LIN {X 0,Y 368.346,Z 298.483,A -85,B 0,C 180,E1 -13235.936,E2 -13235.936} C_VEL
LIN {X 0,Y 372.9,Z 313.274,A -85,B 0,C 180,E1 -13237.03,E2 -13237.03} C_VEL
LIN {X 0,Y 374.658,Z 319.531,A -85,B 0,C 180,E1 -13237.544,E2 -13237.544} C_VEL
LIN {X 0,Y 373.455,Z 332.306,A -85,B 0,C 180,E1 -13238.385,E2 -13238.385} C_VEL
LIN {X 0,Y 371.968,Z 346.016,A -85,B 0,C 180,E1 -13239.515,E2 -13239.515} C_VEL
LIN {X 0,Y 370.336,Z 358.794,A -85,B 0,C 180,E1 -13240.804,E2 -13240.804} C_VEL
LIN {X 0,Y 368.69,Z 371.331,A -85,B 0,C 180,E1 -13242.352,E2 -13242.352} C_VEL
LIN {X 0,Y 366.908,Z 383.259,A -85,B 0,C 180,E1 -13244.135,E2 -13244.135} C_VEL
LIN {X 0,Y 365.422,Z 393.227,A -85,B 0,C 180,E1 -13245.931,E2 -13245.931} C_VEL
LIN {X 0,Y 363.933,Z 402.704,A -85,B 0,C 180,E1 -13247.997,E2 -13247.997} C_VEL
LIN {X 0,Y 362.831,Z 410.613,A -85,B 0,C 180,E1 -13250.109,E2 -13250.109} C_VEL
LIN {X 0,Y 361.936,Z 417.12,A -85,B 0,C 180,E1 -13252.249,E2 -13252.249} C_VEL
LIN {X 0,Y 361.391,Z 421.607,A -85,B 0,C 180,E1 -13254.103,E2 -13254.103} C_VEL
LIN {X 0,Y 360.855,Z 426.279,A -85,B 0,C 180,E1 -13256.611,E2 -13256.611} C_VEL
LIN {X 0,Y 360.458,Z 429.462,A -85,B 0,C 180,E1 -13259.171,E2 -13259.171} C_VEL
LIN {X 0,Y 360.358,Z 430.738,A -85,B 0,C 180,E1 -13260.897,E2 -13260.897} C_VEL
LIN {X 0,Y 360.322,Z 431.406,A -85,B 0,C 180,E1 -13263.101,E2 -13263.101} C_VEL
LIN {X 0,Y 360.359,Z 431.048,A -85,B 0,C 180,E1 -13265.007,E2 -13265.007} C_VEL
LIN {X 0,Y 360.534,Z 429.695,A -85,B 0,C 180,E1 -13267.177,E2 -13267.177} C_VEL
LIN {X 0,Y 360.574,Z 429.284,A -85,B 0,C 180,E1 -13267.57,E2 -13267.57} C_VEL
LIN {X 0,Y 360.044,Z 428.403,A -85,B 0,C 180,E1 -13268.493,E2 -13268.493} C_VEL
LIN {X 0,Y 357.472,Z 426.615,A -85,B 0,C 180,E1 -13269.998,E2 -13269.998} C_VEL
LIN {X 0,Y 355.343,Z 424.907,A -85,B 0,C 180,E1 -13271.203,E2 -13271.203} C_VEL
LIN {X 0,Y 354.556,Z 423.304,A -85,B 0,C 180,E1 -13272.116,E2 -13272.116} C_VEL
LIN {X 0,Y 354.562,Z 422.675,A -85,B 0,C 180,E1 -13272.42,E2 -13272.42} C_VEL
LIN {X 0,Y 355.32,Z 417.558,A -85,B 0,C 180,E1 -13274.6,E2 -13274.6} C_VEL
LIN {X 0,Y 356.455,Z 410.865,A -85,B 0,C 180,E1 -13276.844,E2 -13276.844} C_VEL
LIN {X 0,Y 357.829,Z 402.794,A -85,B 0,C 180,E1 -13279.018,E2 -13279.018} C_VEL
LIN {X 0,Y 359.353,Z 394.035,A -85,B 0,C 180,E1 -13280.959,E2 -13280.959} C_VEL
LIN {X 0,Y 361.095,Z 384.034,A -85,B 0,C 180,E1 -13282.795,E2 -13282.795} C_VEL
LIN {X 0,Y 362.941,Z 372.942,A -85,B 0,C 180,E1 -13284.487,E2 -13284.487} C_VEL
LIN {X 0,Y 364.899,Z 360.545,A -85,B 0,C 180,E1 -13286.047,E2 -13286.047} C_VEL
LIN {X 0,Y 366.644,Z 347.802,A -85,B 0,C 180,E1 -13287.373,E2 -13287.373} C_VEL
LIN {X 0,Y 368.422,Z 333.632,A -85,B 0,C 180,E1 -13288.556,E2 -13288.556} C_VEL
LIN {X 0,Y 369.441,Z 323.375,A -85,B 0,C 180,E1 -13289.254,E2 -13289.254} C_VEL
LIN {X 0,Y 365.365,Z 309.416,A -85,B 0,C 180,E1 -13290.491,E2 -13290.491} C_VEL
LIN {X 0,Y 359.944,Z 295.452,A -85,B 0,C 180,E1 -13291.663,E2 -13291.663} C_VEL
LIN {X 0,Y 355.644,Z 286.065,A -85,B 0,C 180,E1 -13292.411,E2 -13292.411} C_VEL
LIN {X 0,Y 354.613,Z 283.116,A -85,B 0,C 180,E1 -13292.604,E2 -13292.604} C_VEL
LIN {X 0,Y 354.73,Z 280.957,A -85,B 0,C 180,E1 -13295.692,E2 -13295.692} C_VEL
LIN {X 0,Y 354.874,Z 278.678,A -85,B 0,C 180,E1 -13299.118,E2 -13299.118} C_VEL
LIN {X 0,Y 354.894,Z 276.415,A -85,B 0,C 180,E1 -13302.721,E2 -13302.721} C_VEL
LIN {X 0,Y 354.867,Z 275.912,A -85,B 0,C 180,E1 -13303.904,E2 -13303.904} C_VEL
LIN {X 0,Y 354.915,Z 275.902,A -85,B 0,C 180,E1 -13307.42,E2 -13307.42} C_VEL
LIN {X 0,Y 355.122,Z 275.877,A -85,B 0,C 180,E1 -13311.69,E2 -13311.69} C_VEL
LIN {X 0,Y 355.088,Z 275.879,A -85,B 0,C 180,E1 -13314.322,E2 -13314.322} C_VEL
LIN {X 0,Y 355.241,Z 275.859,A -85,B 0,C 180,E1 -13317.734,E2 -13317.734} C_VEL
LIN {X 0,Y 355.393,Z 275.839,A -85,B 0,C 180,E1 -13320.001,E2 -13320.001} C_VEL
LIN {X 0,Y 355.242,Z 275.858,A -85,B 0,C 180,E1 -13322.269,E2 -13322.269} C_VEL
LIN {X 0,Y 355.134,Z 275.873,A -85,B 0,C 180,E1 -13326.82,E2 -13326.82} C_VEL
LIN {X 0,Y 355.011,Z 275.888,A -85,B 0,C 180,E1 -13329.114,E2 -13329.114} C_VEL
LIN {X 0,Y 354.918,Z 275.898,A -85,B 0,C 180,E1 -13332.582,E2 -13332.582} C_VEL
LIN {X 0,Y 354.886,Z 275.904,A -85,B 0,C 180,E1 -13336.097,E2 -13336.097} C_VEL
LIN {X 0,Y 354.903,Z 275.902,A -85,B 0,C 180,E1 -13338.473,E2 -13338.473} C_VEL
LIN {X 0,Y 354.832,Z 275.911,A -85,B 0,C 180,E1 -13342.107,E2 -13342.107} C_VEL
LIN {X 0,Y 354.897,Z 275.902,A -85,B 0,C 180,E1 -13345.829,E2 -13345.829} C_VEL
LIN {X 0,Y 354.852,Z 275.914,A -85,B 0,C 180,E1 -13349.68,E2 -13349.68} C_VEL
LIN {X 0,Y 354.82,Z 276.044,A -85,B 0,C 180,E1 -13352.667,E2 -13352.667} C_VEL
LIN {X 0,Y 355.388,Z 279.05,A -85,B 0,C 180,E1 -13355.828,E2 -13355.828} C_VEL
LIN {X 0,Y 356.119,Z 283.281,A -85,B 0,C 180,E1 -13359.678,E2 -13359.678} C_VEL
LIN {X 0,Y 356.952,Z 288.147,A -85,B 0,C 180,E1 -13363.561,E2 -13363.561} C_VEL
LIN {X 0,Y 357.671,Z 292.442,A -85,B 0,C 180,E1 -13366.639,E2 -13366.639} C_VEL
LIN {X 0,Y 357.676,Z 295.963,A -85,B 0,C 180,E1 -13368.935,E2 -13368.935} C_VEL
LIN {X 0,Y 356.892,Z 301.707,A -85,B 0,C 180,E1 -13372.378,E2 -13372.378} C_VEL
LIN {X 0,Y 356.195,Z 308.035,A -85,B 0,C 180,E1 -13375.966,E2 -13375.966} C_VEL
LIN {X 0,Y 355.518,Z 315.02,A -85,B 0,C 180,E1 -13379.73,E2 -13379.73} C_VEL
LIN {X 0,Y 355.426,Z 316.517,A -85,B 0,C 180,E1 -13380.464,E2 -13380.464} C_VEL
LIN {X 0,Y 356.367,Z 319.81,A -85,B 0,C 180,E1 -13380.638,E2 -13380.638} C_VEL
LIN {X 0,Y 360.801,Z 334.796,A -85,B 0,C 180,E1 -13381.548,E2 -13381.548} C_VEL
LIN {X 0,Y 364.028,Z 349.7,A -85,B 0,C 180,E1 -13382.552,E2 -13382.552} C_VEL
LIN {X 0,Y 366.315,Z 364.769,A -85,B 0,C 180,E1 -13383.695,E2 -13383.695} C_VEL
LIN {X 0,Y 367.111,Z 371.055,A -85,B 0,C 180,E1 -13384.231,E2 -13384.231} C_VEL
LIN {X 0,Y 365.414,Z 384.335,A -85,B 0,C 180,E1 -13385.273,E2 -13385.273} C_VEL
LIN {X 0,Y 363.482,Z 397.146,A -85,B 0,C 180,E1 -13386.498,E2 -13386.498} C_VEL
LIN {X 0,Y 361.493,Z 410.148,A -85,B 0,C 180,E1 -13388.023,E2 -13388.023} C_VEL
LIN {X 0,Y 359.534,Z 422.392,A -85,B 0,C 180,E1 -13389.766,E2 -13389.766} C_VEL
LIN {X 0,Y 357.871,Z 433.506,A -85,B 0,C 180,E1 -13391.688,E2 -13391.688} C_VEL
LIN {X 0,Y 356.341,Z 443.099,A -85,B 0,C 180,E1 -13393.678,E2 -13393.678} C_VEL
LIN {X 0,Y 355.149,Z 451.18,A -85,B 0,C 180,E1 -13395.698,E2 -13395.698} C_VEL
LIN {X 0,Y 354.343,Z 458.64,A -85,B 0,C 180,E1 -13397.981,E2 -13397.981} C_VEL
LIN {X 0,Y 353.715,Z 464.622,A -85,B 0,C 180,E1 -13400.278,E2 -13400.278} C_VEL
LIN {X 0,Y 353.51,Z 468.2,A -85,B 0,C 180,E1 -13402.001,E2 -13402.001} C_VEL
LIN {X 0,Y 353.366,Z 471.82,A -85,B 0,C 180,E1 -13404.294,E2 -13404.294} C_VEL
LIN {X 0,Y 353.27,Z 474.207,A -85,B 0,C 180,E1 -13406.579,E2 -13406.579} C_VEL
LIN {X 0,Y 353.379,Z 475.424,A -85,B 0,C 180,E1 -13408.861,E2 -13408.861} C_VEL
LIN {X 0,Y 353.378,Z 475.45,A -85,B 0,C 180,E1 -13411.14,E2 -13411.14} C_VEL
LIN {X 0,Y 353.261,Z 474.249,A -85,B 0,C 180,E1 -13413.422,E2 -13413.422} C_VEL
LIN {X 0,Y 353.358,Z 471.874,A -85,B 0,C 180,E1 -13415.708,E2 -13415.708} C_VEL
LIN {X 0,Y 353.511,Z 468.264,A -85,B 0,C 180,E1 -13418,E2 -13418} C_VEL
LIN {X 0,Y 353.821,Z 463.331,A -85,B 0,C 180,E1 -13420.299,E2 -13420.299} C_VEL
LIN {X 0,Y 354.511,Z 456.958,A -85,B 0,C 180,E1 -13422.596,E2 -13422.596} C_VEL
LIN {X 0,Y 355.5,Z 448.962,A -85,B 0,C 180,E1 -13424.893,E2 -13424.893} C_VEL
LIN {X 0,Y 356.729,Z 440.46,A -85,B 0,C 180,E1 -13426.894,E2 -13426.894} C_VEL
LIN {X 0,Y 358.097,Z 431.831,A -85,B 0,C 180,E1 -13428.599,E2 -13428.599} C_VEL
LIN {X 0,Y 359.718,Z 420.925,A -85,B 0,C 180,E1 -13430.41,E2 -13430.41} C_VEL
LIN {X 0,Y 361.661,Z 408.477,A -85,B 0,C 180,E1 -13432.118,E2 -13432.118} C_VEL
LIN {X 0,Y 363.565,Z 394.852,A -85,B 0,C 180,E1 -13433.649,E2 -13433.649} C_VEL
LIN {X 0,Y 365.524,Z 381.257,A -85,B 0,C 180,E1 -13434.873,E2 -13434.873} C_VEL
LIN {X 0,Y 366.729,Z 369.526,A -85,B 0,C 180,E1 -13435.748,E2 -13435.748} C_VEL
LIN {X 0,Y 364.294,Z 355.037,A -85,B 0,C 180,E1 -13436.879,E2 -13436.879} C_VEL
LIN {X 0,Y 361.413,Z 340.742,A -85,B 0,C 180,E1 -13437.821,E2 -13437.821} C_VEL
LIN {X 0,Y 357.374,Z 325.464,A -85,B 0,C 180,E1 -13438.689,E2 -13438.689} C_VEL
LIN {X 0,Y 355.389,Z 318.138,A -85,B 0,C 180,E1 -13439.057,E2 -13439.057} C_VEL
LIN {X 0,Y 355.926,Z 312.143,A -85,B 0,C 180,E1 -13442.218,E2 -13442.218} C_VEL
LIN {X 0,Y 356.589,Z 306.081,A -85,B 0,C 180,E1 -13445.488,E2 -13445.488} C_VEL
LIN {X 0,Y 357.325,Z 299.823,A -85,B 0,C 180,E1 -13449.006,E2 -13449.006} C_VEL
LIN {X 0,Y 357.761,Z 294.883,A -85,B 0,C 180,E1 -13451.907,E2 -13451.907} C_VEL
LIN {X 0,Y 357.548,Z 291.222,A -85,B 0,C 180,E1 -13454.2,E2 -13454.2} C_VEL
LIN {X 0,Y 356.56,Z 285.705,A -85,B 0,C 180,E1 -13457.92,E2 -13457.92} C_VEL
LIN {X 0,Y 355.823,Z 281.709,A -85,B 0,C 180,E1 -13460.798,E2 -13460.798} C_VEL
LIN {X 0,Y 355.104,Z 277.225,A -85,B 0,C 180,E1 -13464.238,E2 -13464.238} C_VEL
LIN {X 0,Y 354.843,Z 275.911,A -85,B 0,C 180,E1 -13465.462,E2 -13465.462} C_VEL
LIN {X 0,Y 354.806,Z 275.915,A -85,B 0,C 180,E1 -13469.001,E2 -13469.001} C_VEL
LIN {X 0,Y 354.888,Z 275.905,A -85,B 0,C 180,E1 -13472.903,E2 -13472.903} C_VEL
LIN {X 0,Y 354.867,Z 275.903,A -85,B 0,C 180,E1 -13475.647,E2 -13475.647} C_VEL
LIN {X 0,Y 354.846,Z 275.908,A -85,B 0,C 180,E1 -13479.113,E2 -13479.113} C_VEL
LIN {X 0,Y 354.904,Z 275.904,A -85,B 0,C 180,E1 -13482.719,E2 -13482.719} C_VEL
LIN {X 0,Y 354.957,Z 275.894,A -85,B 0,C 180,E1 -13486.254,E2 -13486.254} C_VEL
LIN {X 0,Y 354.983,Z 275.889,A -85,B 0,C 180,E1 -13489.735,E2 -13489.735} C_VEL
LIN {X 0,Y 355.105,Z 275.874,A -85,B 0,C 180,E1 -13493.179,E2 -13493.179} C_VEL
LIN {X 0,Y 355.248,Z 275.856,A -85,B 0,C 180,E1 -13497.731,E2 -13497.731} C_VEL
LIN {X 0,Y 355.402,Z 275.838,A -85,B 0,C 180,E1 -13499.999,E2 -13499.999} C_VEL
LIN {X 0,Y 355.247,Z 275.86,A -85,B 0,C 180,E1 -13502.266,E2 -13502.266} C_VEL
LIN {X 0,Y 355.142,Z 275.87,A -85,B 0,C 180,E1 -13506.818,E2 -13506.818} C_VEL
LIN {X 0,Y 355.018,Z 275.884,A -85,B 0,C 180,E1 -13509.111,E2 -13509.111} C_VEL
LIN {X 0,Y 354.924,Z 275.898,A -85,B 0,C 180,E1 -13512.579,E2 -13512.579} C_VEL
LIN {X 0,Y 354.892,Z 275.905,A -85,B 0,C 180,E1 -13516.094,E2 -13516.094} C_VEL
LIN {X 0,Y 354.908,Z 275.9,A -85,B 0,C 180,E1 -13518.47,E2 -13518.47} C_VEL
LIN {X 0,Y 354.835,Z 275.912,A -85,B 0,C 180,E1 -13522.104,E2 -13522.104} C_VEL
LIN {X 0,Y 354.899,Z 275.902,A -85,B 0,C 180,E1 -13525.826,E2 -13525.826} C_VEL
LIN {X 0,Y 354.816,Z 275.911,A -85,B 0,C 180,E1 -13529.68,E2 -13529.68} C_VEL
LIN {X 0,Y 354.804,Z 275.914,A -85,B 0,C 180,E1 -13533.7,E2 -13533.7} C_VEL
LIN {X 0,Y 354.796,Z 275.913,A -85,B 0,C 180,E1 -13536.458,E2 -13536.458} C_VEL
LIN {X 0,Y 354.821,Z 275.91,A -85,B 0,C 180,E1 -13539.422,E2 -13539.422} C_VEL
LIN {X 0,Y 354.788,Z 275.912,A -85,B 0,C 180,E1 -13542.866,E2 -13542.866} C_VEL
LIN {X 0,Y 354.848,Z 275.908,A -85,B 0,C 180,E1 -13546.115,E2 -13546.115} C_VEL
LIN {X 0,Y 354.852,Z 275.905,A -85,B 0,C 180,E1 -13549.187,E2 -13549.187} C_VEL
LIN {X 0,Y 354.803,Z 275.911,A -85,B 0,C 180,E1 -13552.401,E2 -13552.401} C_VEL
LIN {X 0,Y 354.806,Z 275.91,A -85,B 0,C 180,E1 -13554.939,E2 -13554.939} C_VEL
LIN {X 0,Y 354.786,Z 275.913,A -85,B 0,C 180,E1 -13558.404,E2 -13558.404} C_VEL
LIN {X 0,Y 354.846,Z 275.912,A -85,B 0,C 180,E1 -13561.618,E2 -13561.618} C_VEL
LIN {X 0,Y 354.891,Z 275.901,A -85,B 0,C 180,E1 -13564.171,E2 -13564.171} C_VEL
LIN {X 0,Y 354.826,Z 275.91,A -85,B 0,C 180,E1 -13567.893,E2 -13567.893} C_VEL
LIN {X 0,Y 354.914,Z 275.899,A -85,B 0,C 180,E1 -13571.89,E2 -13571.89} C_VEL
LIN {X 0,Y 354.934,Z 275.896,A -85,B 0,C 180,E1 -13575.98,E2 -13575.98} C_VEL
LIN {X 0,Y 354.973,Z 275.892,A -85,B 0,C 180,E1 -13579.735,E2 -13579.735} C_VEL
LIN {X 0,Y 355.103,Z 275.873,A -85,B 0,C 180,E1 -13582.036,E2 -13582.036} C_VEL
LIN {X 0,Y 355.066,Z 275.878,A -85,B 0,C 180,E1 -13584.32,E2 -13584.32} C_VEL
LIN {X 0,Y 355.015,Z 276.113,A -85,B 0,C 180,E1 -13588.865,E2 -13588.865} C_VEL
LIN {X 0,Y 354.385,Z 280.472,A -85,B 0,C 180,E1 -13594.193,E2 -13594.193} C_VEL
LIN {X 0,Y 356.694,Z 286.53,A -85,B 0,C 180,E1 -13594.558,E2 -13594.558} C_VEL
LIN {X 0,Y 362.27,Z 301.422,A -85,B 0,C 180,E1 -13595.587,E2 -13595.587} C_VEL
LIN {X 0,Y 366.282,Z 314.648,A -85,B 0,C 180,E1 -13596.61,E2 -13596.61} C_VEL
LIN {X 0,Y 368.088,Z 321.326,A -85,B 0,C 180,E1 -13597.179,E2 -13597.179} C_VEL
LIN {X 0,Y 366.7,Z 334.988,A -85,B 0,C 180,E1 -13598.125,E2 -13598.125} C_VEL
LIN {X 0,Y 365.203,Z 348.245,A -85,B 0,C 180,E1 -13599.274,E2 -13599.274} C_VEL
LIN {X 0,Y 363.578,Z 360.207,A -85,B 0,C 180,E1 -13600.524,E2 -13600.524} C_VEL
LIN {X 0,Y 361.934,Z 372.216,A -85,B 0,C 180,E1 -13602.048,E2 -13602.048} C_VEL
LIN {X 0,Y 360.447,Z 382.067,A -85,B 0,C 180,E1 -13603.53,E2 -13603.53} C_VEL
LIN {X 0,Y 358.81,Z 392.168,A -85,B 0,C 180,E1 -13605.332,E2 -13605.332} C_VEL
LIN {X 0,Y 357.39,Z 400.719,A -85,B 0,C 180,E1 -13607.155,E2 -13607.155} C_VEL
LIN {X 0,Y 356.256,Z 408.565,A -85,B 0,C 180,E1 -13609.166,E2 -13609.166} C_VEL
LIN {X 0,Y 355.443,Z 414.117,A -85,B 0,C 180,E1 -13610.848,E2 -13610.848} C_VEL
LIN {X 0,Y 354.704,Z 419.222,A -85,B 0,C 180,E1 -13612.728,E2 -13612.728} C_VEL
LIN {X 0,Y 354.179,Z 423.45,A -85,B 0,C 180,E1 -13614.626,E2 -13614.626} C_VEL
LIN {X 0,Y 353.78,Z 426.91,A -85,B 0,C 180,E1 -13616.631,E2 -13616.631} C_VEL
LIN {X 0,Y 353.408,Z 429.74,A -85,B 0,C 180,E1 -13618.959,E2 -13618.959} C_VEL
LIN {X 0,Y 353.273,Z 431.32,A -85,B 0,C 180,E1 -13621.195,E2 -13621.195} C_VEL
LIN {X 0,Y 353.226,Z 431.845,A -85,B 0,C 180,E1 -13623.319,E2 -13623.319} C_VEL
LIN {X 0,Y 353.284,Z 431.388,A -85,B 0,C 180,E1 -13625.354,E2 -13625.354} C_VEL
LIN {X 0,Y 353.575,Z 429.439,A -85,B 0,C 180,E1 -13628.037,E2 -13628.037} C_VEL
LIN {X 0,Y 353.97,Z 426.681,A -85,B 0,C 180,E1 -13630.185,E2 -13630.185} C_VEL
LIN {X 0,Y 354.562,Z 422.675,A -85,B 0,C 180,E1 -13632.42,E2 -13632.42} C_VEL
LIN {X 0,Y 354.187,Z 420.817,A -85,B 0,C 180,E1 -13633.324,E2 -13633.324} C_VEL
LIN {X 0,Y 351.901,Z 417.626,A -85,B 0,C 180,E1 -13634.804,E2 -13634.804} C_VEL
LIN {X 0,Y 349.743,Z 413.979,A -85,B 0,C 180,E1 -13636.27,E2 -13636.27} C_VEL
LIN {X 0,Y 349.567,Z 411.346,A -85,B 0,C 180,E1 -13637.137,E2 -13637.137} C_VEL
LIN {X 0,Y 350.959,Z 403.72,A -85,B 0,C 180,E1 -13639.25,E2 -13639.25} C_VEL
LIN {X 0,Y 352.567,Z 394.833,A -85,B 0,C 180,E1 -13641.271,E2 -13641.271} C_VEL
LIN {X 0,Y 354.314,Z 385.25,A -85,B 0,C 180,E1 -13643.079,E2 -13643.079} C_VEL
LIN {X 0,Y 356.349,Z 373.692,A -85,B 0,C 180,E1 -13644.89,E2 -13644.89} C_VEL
LIN {X 0,Y 358.349,Z 361.629,A -85,B 0,C 180,E1 -13646.446,E2 -13646.446} C_VEL
LIN {X 0,Y 360.282,Z 348.202,A -85,B 0,C 180,E1 -13647.871,E2 -13647.871} C_VEL
LIN {X 0,Y 362.13,Z 334.183,A -85,B 0,C 180,E1 -13649.058,E2 -13649.058} C_VEL
LIN {X 0,Y 362.94,Z 326.406,A -85,B 0,C 180,E1 -13649.612,E2 -13649.612} C_VEL
LIN {X 0,Y 362.56,Z 323.397,A -85,B 0,C 180,E1 -13649.863,E2 -13649.863} C_VEL
LIN {X 0,Y 358.992,Z 311.346,A -85,B 0,C 180,E1 -13650.983,E2 -13650.983} C_VEL
LIN {X 0,Y 354.258,Z 298.775,A -85,B 0,C 180,E1 -13652.093,E2 -13652.093} C_VEL
LIN {X 0,Y 349.013,Z 287.122,A -85,B 0,C 180,E1 -13653.067,E2 -13653.067} C_VEL
LIN {X 0,Y 347.779,Z 284.415,A -85,B 0,C 180,E1 -13653.285,E2 -13653.285} C_VEL
LIN {X 0,Y 347.631,Z 283.617,A -85,B 0,C 180,E1 -13653.353,E2 -13653.353} C_VEL
LIN {X 0,Y 347.713,Z 281.728,A -85,B 0,C 180,E1 -13656.158,E2 -13656.158} C_VEL
LIN {X 0,Y 347.854,Z 280.077,A -85,B 0,C 180,E1 -13658.676,E2 -13658.676} C_VEL
LIN {X 0,Y 347.901,Z 277.805,A -85,B 0,C 180,E1 -13662.363,E2 -13662.363} C_VEL
LIN {X 0,Y 347.853,Z 276.785,A -85,B 0,C 180,E1 -13664.774,E2 -13664.774} C_VEL
LIN {X 0,Y 347.878,Z 276.778,A -85,B 0,C 180,E1 -13668.346,E2 -13668.346} C_VEL
LIN {X 0,Y 348.068,Z 276.756,A -85,B 0,C 180,E1 -13671.876,E2 -13671.876} C_VEL
LIN {X 0,Y 348.063,Z 276.754,A -85,B 0,C 180,E1 -13674.207,E2 -13674.207} C_VEL
LIN {X 0,Y 348.204,Z 276.735,A -85,B 0,C 180,E1 -13677.688,E2 -13677.688} C_VEL
LIN {X 0,Y 348.342,Z 276.717,A -85,B 0,C 180,E1 -13680.001,E2 -13680.001} C_VEL
LIN {X 0,Y 348.204,Z 276.735,A -85,B 0,C 180,E1 -13682.315,E2 -13682.315} C_VEL
LIN {X 0,Y 348.103,Z 276.749,A -85,B 0,C 180,E1 -13686.959,E2 -13686.959} C_VEL
LIN {X 0,Y 347.964,Z 276.767,A -85,B 0,C 180,E1 -13689.3,E2 -13689.3} C_VEL
LIN {X 0,Y 347.887,Z 276.772,A -85,B 0,C 180,E1 -13692.841,E2 -13692.841} C_VEL
LIN {X 0,Y 347.836,Z 276.782,A -85,B 0,C 180,E1 -13696.433,E2 -13696.433} C_VEL
LIN {X 0,Y 347.853,Z 276.779,A -85,B 0,C 180,E1 -13698.861,E2 -13698.861} C_VEL
LIN {X 0,Y 347.772,Z 276.792,A -85,B 0,C 180,E1 -13702.581,E2 -13702.581} C_VEL
LIN {X 0,Y 347.81,Z 276.784,A -85,B 0,C 180,E1 -13705.11,E2 -13705.11} C_VEL
LIN {X 0,Y 347.809,Z 276.787,A -85,B 0,C 180,E1 -13707.695,E2 -13707.695} C_VEL
LIN {X 0,Y 347.762,Z 276.796,A -85,B 0,C 180,E1 -13710.348,E2 -13710.348} C_VEL
LIN {X 0,Y 347.797,Z 277.037,A -85,B 0,C 180,E1 -13711.931,E2 -13711.931} C_VEL
LIN {X 0,Y 348.458,Z 280.588,A -85,B 0,C 180,E1 -13715.797,E2 -13715.797} C_VEL
LIN {X 0,Y 348.956,Z 283.6,A -85,B 0,C 180,E1 -13718.635,E2 -13718.635} C_VEL
LIN {X 0,Y 349.619,Z 287.493,A -85,B 0,C 180,E1 -13721.948,E2 -13721.948} C_VEL
LIN {X 0,Y 350.464,Z 292.031,A -85,B 0,C 180,E1 -13725.424,E2 -13725.424} C_VEL
LIN {X 0,Y 350.758,Z 295.538,A -85,B 0,C 180,E1 -13727.848,E2 -13727.848} C_VEL
LIN {X 0,Y 350.227,Z 300.199,A -85,B 0,C 180,E1 -13730.795,E2 -13730.795} C_VEL
LIN {X 0,Y 349.499,Z 306.156,A -85,B 0,C 180,E1 -13734.328,E2 -13734.328} C_VEL
LIN {X 0,Y 348.775,Z 312.345,A -85,B 0,C 180,E1 -13737.815,E2 -13737.815} C_VEL
LIN {X 0,Y 348.47,Z 315.987,A -85,B 0,C 180,E1 -13739.748,E2 -13739.748} C_VEL
LIN {X 0,Y 349.445,Z 319.338,A -85,B 0,C 180,E1 -13739.938,E2 -13739.938} C_VEL
LIN {X 0,Y 354.287,Z 335.29,A -85,B 0,C 180,E1 -13740.973,E2 -13740.973} C_VEL
LIN {X 0,Y 357.541,Z 350.356,A -85,B 0,C 180,E1 -13742.031,E2 -13742.031} C_VEL
LIN {X 0,Y 359.836,Z 366.392,A -85,B 0,C 180,E1 -13743.308,E2 -13743.308} C_VEL
LIN {X 0,Y 360.556,Z 372.164,A -85,B 0,C 180,E1 -13743.823,E2 -13743.823} C_VEL
LIN {X 0,Y 358.716,Z 385.725,A -85,B 0,C 180,E1 -13744.934,E2 -13744.934} C_VEL
LIN {X 0,Y 356.54,Z 399.492,A -85,B 0,C 180,E1 -13746.321,E2 -13746.321} C_VEL
LIN {X 0,Y 354.483,Z 412.02,A -85,B 0,C 180,E1 -13747.872,E2 -13747.872} C_VEL
LIN {X 0,Y 352.44,Z 424.352,A -85,B 0,C 180,E1 -13749.725,E2 -13749.725} C_VEL
LIN {X 0,Y 350.789,Z 434.671,A -85,B 0,C 180,E1 -13751.607,E2 -13751.607} C_VEL
LIN {X 0,Y 349.275,Z 443.978,A -85,B 0,C 180,E1 -13753.639,E2 -13753.639} C_VEL
LIN {X 0,Y 347.964,Z 452.21,A -85,B 0,C 180,E1 -13755.81,E2 -13755.81} C_VEL
LIN {X 0,Y 347.32,Z 458.229,A -85,B 0,C 180,E1 -13757.734,E2 -13757.734} C_VEL
LIN {X 0,Y 346.657,Z 464.204,A -85,B 0,C 180,E1 -13760.078,E2 -13760.078} C_VEL
LIN {X 0,Y 346.43,Z 467.782,A -85,B 0,C 180,E1 -13761.837,E2 -13761.837} C_VEL
LIN {X 0,Y 346.291,Z 471.396,A -85,B 0,C 180,E1 -13764.177,E2 -13764.177} C_VEL
LIN {X 0,Y 346.192,Z 473.777,A -85,B 0,C 180,E1 -13766.509,E2 -13766.509} C_VEL
LIN {X 0,Y 346.301,Z 474.987,A -85,B 0,C 180,E1 -13768.838,E2 -13768.838} C_VEL
LIN {X 0,Y 346.301,Z 475.011,A -85,B 0,C 180,E1 -13771.164,E2 -13771.164} C_VEL
LIN {X 0,Y 346.184,Z 473.799,A -85,B 0,C 180,E1 -13773.492,E2 -13773.492} C_VEL
LIN {X 0,Y 346.328,Z 471.085,A -85,B 0,C 180,E1 -13776.087,E2 -13776.087} C_VEL
LIN {X 0,Y 346.499,Z 466.706,A -85,B 0,C 180,E1 -13778.751,E2 -13778.751} C_VEL
LIN {X 0,Y 346.951,Z 461.396,A -85,B 0,C 180,E1 -13781.096,E2 -13781.096} C_VEL
LIN {X 0,Y 347.726,Z 454.615,A -85,B 0,C 180,E1 -13783.441,E2 -13783.441} C_VEL
LIN {X 0,Y 348.718,Z 447.312,A -85,B 0,C 180,E1 -13785.489,E2 -13785.489} C_VEL
LIN {X 0,Y 350.024,Z 438.551,A -85,B 0,C 180,E1 -13787.529,E2 -13787.529} C_VEL
LIN {X 0,Y 351.806,Z 428.034,A -85,B 0,C 180,E1 -13789.55,E2 -13789.55} C_VEL
LIN {X 0,Y 353.456,Z 417.252,A -85,B 0,C 180,E1 -13791.278,E2 -13791.278} C_VEL
LIN {X 0,Y 355.535,Z 404.358,A -85,B 0,C 180,E1 -13792.98,E2 -13792.98} C_VEL
LIN {X 0,Y 357.427,Z 391.353,A -85,B 0,C 180,E1 -13794.389,E2 -13794.389} C_VEL
LIN {X 0,Y 359.477,Z 377.334,A -85,B 0,C 180,E1 -13795.606,E2 -13795.606} C_VEL
LIN {X 0,Y 360.05,Z 370.656,A -85,B 0,C 180,E1 -13796.116,E2 -13796.116} C_VEL
LIN {X 0,Y 357.61,Z 355.6,A -85,B 0,C 180,E1 -13797.33,E2 -13797.33} C_VEL
LIN {X 0,Y 354.727,Z 341.278,A -85,B 0,C 180,E1 -13798.314,E2 -13798.314} C_VEL
LIN {X 0,Y 350.734,Z 326.146,A -85,B 0,C 180,E1 -13799.217,E2 -13799.217} C_VEL
LIN {X 0,Y 348.459,Z 317.743,A -85,B 0,C 180,E1 -13799.658,E2 -13799.658} C_VEL
LIN {X 0,Y 349.017,Z 311.668,A -85,B 0,C 180,E1 -13802.936,E2 -13802.936} C_VEL
LIN {X 0,Y 349.738,Z 305.25,A -85,B 0,C 180,E1 -13806.504,E2 -13806.504} C_VEL
LIN {X 0,Y 350.464,Z 299.368,A -85,B 0,C 180,E1 -13809.92,E2 -13809.92} C_VEL
LIN {X 0,Y 350.774,Z 295.644,A -85,B 0,C 180,E1 -13812.155,E2 -13812.155} C_VEL
LIN {X 0,Y 350.482,Z 291.891,A -85,B 0,C 180,E1 -13814.575,E2 -13814.575} C_VEL
LIN {X 0,Y 349.473,Z 286.351,A -85,B 0,C 180,E1 -13818.421,E2 -13818.421} C_VEL
LIN {X 0,Y 348.638,Z 281.792,A -85,B 0,C 180,E1 -13821.831,E2 -13821.831} C_VEL
LIN {X 0,Y 348.18,Z 278.799,A -85,B 0,C 180,E1 -13824.17,E2 -13824.17} C_VEL
LIN {X 0,Y 347.79,Z 276.788,A -85,B 0,C 180,E1 -13825.947,E2 -13825.947} C_VEL
LIN {X 0,Y 347.755,Z 276.79,A -85,B 0,C 180,E1 -13829.652,E2 -13829.652} C_VEL
LIN {X 0,Y 347.837,Z 276.779,A -85,B 0,C 180,E1 -13833.607,E2 -13833.607} C_VEL
LIN {X 0,Y 347.795,Z 276.786,A -85,B 0,C 180,E1 -13836.161,E2 -13836.161} C_VEL
LIN {X 0,Y 347.819,Z 276.781,A -85,B 0,C 180,E1 -13839.909,E2 -13839.909} C_VEL
LIN {X 0,Y 347.872,Z 276.778,A -85,B 0,C 180,E1 -13842.359,E2 -13842.359} C_VEL
LIN {X 0,Y 347.903,Z 276.771,A -85,B 0,C 180,E1 -13845.97,E2 -13845.97} C_VEL
LIN {X 0,Y 347.934,Z 276.767,A -85,B 0,C 180,E1 -13849.525,E2 -13849.525} C_VEL
LIN {X 0,Y 348.073,Z 276.751,A -85,B 0,C 180,E1 -13853.041,E2 -13853.041} C_VEL
LIN {X 0,Y 348.211,Z 276.732,A -85,B 0,C 180,E1 -13857.685,E2 -13857.685} C_VEL
LIN {X 0,Y 348.351,Z 276.717,A -85,B 0,C 180,E1 -13859.999,E2 -13859.999} C_VEL
LIN {X 0,Y 348.209,Z 276.738,A -85,B 0,C 180,E1 -13862.312,E2 -13862.312} C_VEL
LIN {X 0,Y 348.11,Z 276.745,A -85,B 0,C 180,E1 -13866.956,E2 -13866.956} C_VEL
LIN {X 0,Y 347.971,Z 276.762,A -85,B 0,C 180,E1 -13869.297,E2 -13869.297} C_VEL
LIN {X 0,Y 347.893,Z 276.772,A -85,B 0,C 180,E1 -13872.838,E2 -13872.838} C_VEL
LIN {X 0,Y 347.841,Z 276.782,A -85,B 0,C 180,E1 -13876.43,E2 -13876.43} C_VEL
LIN {X 0,Y 347.857,Z 276.776,A -85,B 0,C 180,E1 -13878.859,E2 -13878.859} C_VEL
LIN {X 0,Y 347.775,Z 276.788,A -85,B 0,C 180,E1 -13882.578,E2 -13882.578} C_VEL
LIN {X 0,Y 347.812,Z 276.782,A -85,B 0,C 180,E1 -13885.107,E2 -13885.107} C_VEL
LIN {X 0,Y 347.807,Z 276.784,A -85,B 0,C 180,E1 -13887.692,E2 -13887.692} C_VEL
LIN {X 0,Y 347.748,Z 276.792,A -85,B 0,C 180,E1 -13890.346,E2 -13890.346} C_VEL
LIN {X 0,Y 347.746,Z 276.794,A -85,B 0,C 180,E1 -13894.042,E2 -13894.042} C_VEL
LIN {X 0,Y 347.76,Z 276.788,A -85,B 0,C 180,E1 -13897.319,E2 -13897.319} C_VEL
LIN {X 0,Y 347.73,Z 276.794,A -85,B 0,C 180,E1 -13900.295,E2 -13900.295} C_VEL
LIN {X 0,Y 347.743,Z 276.791,A -85,B 0,C 180,E1 -13903.403,E2 -13903.403} C_VEL
LIN {X 0,Y 347.781,Z 276.786,A -85,B 0,C 180,E1 -13906.674,E2 -13906.674} C_VEL
LIN {X 0,Y 347.78,Z 276.788,A -85,B 0,C 180,E1 -13910.164,E2 -13910.164} C_VEL
LIN {X 0,Y 347.783,Z 276.787,A -85,B 0,C 180,E1 -13914.123,E2 -13914.123} C_VEL
LIN {X 0,Y 347.732,Z 276.794,A -85,B 0,C 180,E1 -13918.085,E2 -13918.085} C_VEL
LIN {X 0,Y 347.799,Z 276.784,A -85,B 0,C 180,E1 -13920.989,E2 -13920.989} C_VEL
LIN {X 0,Y 347.825,Z 276.786,A -85,B 0,C 180,E1 -13923.606,E2 -13923.606} C_VEL
LIN {X 0,Y 347.78,Z 276.787,A -85,B 0,C 180,E1 -13926.161,E2 -13926.161} C_VEL
LIN {X 0,Y 347.808,Z 276.785,A -85,B 0,C 180,E1 -13929.908,E2 -13929.908} C_VEL
LIN {X 0,Y 347.857,Z 276.776,A -85,B 0,C 180,E1 -13932.358,E2 -13932.358} C_VEL
LIN {X 0,Y 347.888,Z 276.774,A -85,B 0,C 180,E1 -13935.97,E2 -13935.97} C_VEL
LIN {X 0,Y 347.923,Z 276.773,A -85,B 0,C 180,E1 -13939.525,E2 -13939.525} C_VEL
LIN {X 0,Y 348.063,Z 276.75,A -85,B 0,C 180,E1 -13941.874,E2 -13941.874} C_VEL
LIN {X 0,Y 348.043,Z 276.753,A -85,B 0,C 180,E1 -13944.205,E2 -13944.205} C_VEL
LIN {X 0,Y 347.631,Z 276.81,A -85,B 0,C 180,E1 -13947.682,E2 -13947.682} C_VEL
LIN {X 0,Y 347.977,Z 277.04,A -85,B 0,C 180,E1 -13948.842,E2 -13948.842} C_VEL
LIN {X 0,Y 347.265,Z 280.808,A -85,B 0,C 180,E1 -13953.58,E2 -13953.58} C_VEL
LIN {X 0,Y 348.264,Z 283.781,A -85,B 0,C 180,E1 -13953.757,E2 -13953.757} C_VEL
LIN {X 0,Y 352.369,Z 293.8,A -85,B 0,C 180,E1 -13954.448,E2 -13954.448} C_VEL
LIN {X 0,Y 357.06,Z 307.165,A -85,B 0,C 180,E1 -13955.456,E2 -13955.456} C_VEL
LIN {X 0,Y 361.301,Z 321.928,A -85,B 0,C 180,E1 -13956.702,E2 -13956.702} C_VEL
LIN {X 0,Y 361.554,Z 322.763,A -85,B 0,C 180,E1 -13956.779,E2 -13956.779} C_VEL
LIN {X 0,Y 360.179,Z 335.795,A -85,B 0,C 180,E1 -13957.708,E2 -13957.708} C_VEL
LIN {X 0,Y 358.62,Z 348.994,A -85,B 0,C 180,E1 -13958.877,E2 -13958.877} C_VEL
LIN {X 0,Y 356.851,Z 361.409,A -85,B 0,C 180,E1 -13960.209,E2 -13960.209} C_VEL
LIN {X 0,Y 355.211,Z 372.886,A -85,B 0,C 180,E1 -13961.7,E2 -13961.7} C_VEL
LIN {X 0,Y 353.472,Z 383.783,A -85,B 0,C 180,E1 -13963.387,E2 -13963.387} C_VEL
LIN {X 0,Y 351.748,Z 394.238,A -85,B 0,C 180,E1 -13965.338,E2 -13965.338} C_VEL
LIN {X 0,Y 350.307,Z 402.623,A -85,B 0,C 180,E1 -13967.212,E2 -13967.212} C_VEL
LIN {X 0,Y 349.059,Z 410.825,A -85,B 0,C 180,E1 -13969.441,E2 -13969.441} C_VEL
LIN {X 0,Y 347.989,Z 417.608,A -85,B 0,C 180,E1 -13971.723,E2 -13971.723} C_VEL
LIN {X 0,Y 347.172,Z 423.675,A -85,B 0,C 180,E1 -13974.366,E2 -13974.366} C_VEL
LIN {X 0,Y 346.659,Z 427.855,A -85,B 0,C 180,E1 -13976.874,E2 -13976.874} C_VEL
LIN {X 0,Y 346.307,Z 430.512,A -85,B 0,C 180,E1 -13979.236,E2 -13979.236} C_VEL
LIN {X 0,Y 346.168,Z 432.061,A -85,B 0,C 180,E1 -13981.86,E2 -13981.86} C_VEL
LIN {X 0,Y 346.138,Z 432.258,A -85,B 0,C 180,E1 -13983.651,E2 -13983.651} C_VEL
LIN {X 0,Y 346.259,Z 431.528,A -85,B 0,C 180,E1 -13986.057,E2 -13986.057} C_VEL
LIN {X 0,Y 346.447,Z 430.3,A -85,B 0,C 180,E1 -13987.71,E2 -13987.71} C_VEL
LIN {X 0,Y 346.798,Z 428.177,A -85,B 0,C 180,E1 -13989.641,E2 -13989.641} C_VEL
LIN {X 0,Y 347.344,Z 424.588,A -85,B 0,C 180,E1 -13991.889,E2 -13991.889} C_VEL
LIN {X 0,Y 348.081,Z 419.777,A -85,B 0,C 180,E1 -13994.152,E2 -13994.152} C_VEL
LIN {X 0,Y 349.162,Z 413.557,A -85,B 0,C 180,E1 -13996.435,E2 -13996.435} C_VEL
LIN {X 0,Y 349.567,Z 411.346,A -85,B 0,C 180,E1 -13997.137,E2 -13997.137} C_VEL
LIN {X 0,Y 349.446,Z 408.605,A -85,B 0,C 180,E1 -13997.993,E2 -13997.993} C_VEL
LIN {X 0,Y 347.595,Z 404.04,A -85,B 0,C 180,E1 -13999.412,E2 -13999.412} C_VEL
LIN {X 0,Y 345.813,Z 399.075,A -85,B 0,C 180,E1 -14000.802,E2 -14000.802} C_VEL
LIN {X 0,Y 345.791,Z 395.621,A -85,B 0,C 180,E1 -14001.597,E2 -14001.597} C_VEL
LIN {X 0,Y 347.719,Z 385.774,A -85,B 0,C 180,E1 -14003.497,E2 -14003.497} C_VEL
LIN {X 0,Y 349.716,Z 374.761,A -85,B 0,C 180,E1 -14005.262,E2 -14005.262} C_VEL
LIN {X 0,Y 351.778,Z 362.922,A -85,B 0,C 180,E1 -14006.83,E2 -14006.83} C_VEL
LIN {X 0,Y 353.747,Z 349.991,A -85,B 0,C 180,E1 -14008.247,E2 -14008.247} C_VEL
LIN {X 0,Y 355.595,Z 336.755,A -85,B 0,C 180,E1 -14009.419,E2 -14009.419} C_VEL
LIN {X 0,Y 356.653,Z 327.452,A -85,B 0,C 180,E1 -14010.115,E2 -14010.115} C_VEL
LIN {X 0,Y 354.333,Z 318.213,A -85,B 0,C 180,E1 -14011.004,E2 -14011.004} C_VEL
LIN {X 0,Y 349.469,Z 304.35,A -85,B 0,C 180,E1 -14012.313,E2 -14012.313} C_VEL
LIN {X 0,Y 343.892,Z 291.349,A -85,B 0,C 180,E1 -14013.488,E2 -14013.488} C_VEL
LIN {X 0,Y 340.879,Z 285.382,A -85,B 0,C 180,E1 -14014.018,E2 -14014.018} C_VEL
LIN {X 0,Y 340.59,Z 284.169,A -85,B 0,C 180,E1 -14014.117,E2 -14014.117} C_VEL
LIN {X 0,Y 340.715,Z 282.328,A -85,B 0,C 180,E1 -14016.928,E2 -14016.928} C_VEL
LIN {X 0,Y 340.856,Z 280.723,A -85,B 0,C 180,E1 -14019.483,E2 -14019.483} C_VEL
LIN {X 0,Y 340.916,Z 279.209,A -85,B 0,C 180,E1 -14021.989,E2 -14021.989} C_VEL
LIN {X 0,Y 340.813,Z 277.813,A -85,B 0,C 180,E1 -14024.452,E2 -14024.452} C_VEL
LIN {X 0,Y 340.837,Z 277.655,A -85,B 0,C 180,E1 -14026.892,E2 -14026.892} C_VEL
LIN {X 0,Y 340.922,Z 277.646,A -85,B 0,C 180,E1 -14030.509,E2 -14030.509} C_VEL
LIN {X 0,Y 341.07,Z 277.625,A -85,B 0,C 180,E1 -14032.899,E2 -14032.899} C_VEL
LIN {X 0,Y 341.165,Z 277.612,A -85,B 0,C 180,E1 -14037.64,E2 -14037.64} C_VEL
LIN {X 0,Y 341.292,Z 277.595,A -85,B 0,C 180,E1 -14040.001,E2 -14040.001} C_VEL
LIN {X 0,Y 341.166,Z 277.612,A -85,B 0,C 180,E1 -14042.362,E2 -14042.362} C_VEL
LIN {X 0,Y 341.072,Z 277.626,A -85,B 0,C 180,E1 -14047.103,E2 -14047.103} C_VEL
LIN {X 0,Y 340.867,Z 277.647,A -85,B 0,C 180,E1 -14050.695,E2 -14050.695} C_VEL
LIN {X 0,Y 340.86,Z 277.651,A -85,B 0,C 180,E1 -14054.326,E2 -14054.326} C_VEL
LIN {X 0,Y 340.835,Z 277.655,A -85,B 0,C 180,E1 -14058.468,E2 -14058.468} C_VEL
LIN {X 0,Y 340.751,Z 277.663,A -85,B 0,C 180,E1 -14061.858,E2 -14061.858} C_VEL
LIN {X 0,Y 340.77,Z 277.661,A -85,B 0,C 180,E1 -14065.666,E2 -14065.666} C_VEL
LIN {X 0,Y 340.739,Z 277.671,A -85,B 0,C 180,E1 -14068.321,E2 -14068.321} C_VEL
LIN {X 0,Y 340.751,Z 277.944,A -85,B 0,C 180,E1 -14071.04,E2 -14071.04} C_VEL
LIN {X 0,Y 341.327,Z 280.964,A -85,B 0,C 180,E1 -14074.554,E2 -14074.554} C_VEL
LIN {X 0,Y 341.908,Z 284.498,A -85,B 0,C 180,E1 -14078.073,E2 -14078.073} C_VEL
LIN {X 0,Y 342.467,Z 287.871,A -85,B 0,C 180,E1 -14081.049,E2 -14081.049} C_VEL
LIN {X 0,Y 343.208,Z 291.805,A -85,B 0,C 180,E1 -14084.218,E2 -14084.218} C_VEL
LIN {X 0,Y 343.724,Z 295.182,A -85,B 0,C 180,E1 -14086.735,E2 -14086.735} C_VEL
LIN {X 0,Y 343.573,Z 298.824,A -85,B 0,C 180,E1 -14089.189,E2 -14089.189} C_VEL
LIN {X 0,Y 342.711,Z 305.138,A -85,B 0,C 180,E1 -14093.11,E2 -14093.11} C_VEL
LIN {X 0,Y 341.902,Z 311.702,A -85,B 0,C 180,E1 -14096.942,E2 -14096.942} C_VEL
LIN {X 0,Y 341.563,Z 315.312,A -85,B 0,C 180,E1 -14098.979,E2 -14098.979} C_VEL
LIN {X 0,Y 342.519,Z 318.815,A -85,B 0,C 180,E1 -14099.196,E2 -14099.196} C_VEL
LIN {X 0,Y 346.852,Z 332.456,A -85,B 0,C 180,E1 -14100.128,E2 -14100.128} C_VEL
LIN {X 0,Y 350.16,Z 346.422,A -85,B 0,C 180,E1 -14101.146,E2 -14101.146} C_VEL
LIN {X 0,Y 352.531,Z 361.131,A -85,B 0,C 180,E1 -14102.309,E2 -14102.309} C_VEL
LIN {X 0,Y 354.029,Z 373.363,A -85,B 0,C 180,E1 -14103.408,E2 -14103.408} C_VEL
LIN {X 0,Y 352.036,Z 387.111,A -85,B 0,C 180,E1 -14104.583,E2 -14104.583} C_VEL
LIN {X 0,Y 349.795,Z 400.503,A -85,B 0,C 180,E1 -14105.993,E2 -14105.993} C_VEL
LIN {X 0,Y 347.664,Z 412.778,A -85,B 0,C 180,E1 -14107.571,E2 -14107.571} C_VEL
LIN {X 0,Y 345.58,Z 424.782,A -85,B 0,C 180,E1 -14109.444,E2 -14109.444} C_VEL
LIN {X 0,Y 344.001,Z 434.338,A -85,B 0,C 180,E1 -14111.231,E2 -14111.231} C_VEL
LIN {X 0,Y 342.375,Z 443.624,A -85,B 0,C 180,E1 -14113.3,E2 -14113.3} C_VEL
LIN {X 0,Y 341.106,Z 451.376,A -85,B 0,C 180,E1 -14115.382,E2 -14115.382} C_VEL
LIN {X 0,Y 340.307,Z 457.833,A -85,B 0,C 180,E1 -14117.477,E2 -14117.477} C_VEL
LIN {X 0,Y 339.614,Z 463.792,A -85,B 0,C 180,E1 -14119.87,E2 -14119.87} C_VEL
LIN {X 0,Y 339.367,Z 467.365,A -85,B 0,C 180,E1 -14121.666,E2 -14121.666} C_VEL
LIN {X 0,Y 339.212,Z 470.973,A -85,B 0,C 180,E1 -14124.055,E2 -14124.055} C_VEL
LIN {X 0,Y 339.116,Z 473.348,A -85,B 0,C 180,E1 -14126.436,E2 -14126.436} C_VEL
LIN {X 0,Y 339.21,Z 474.55,A -85,B 0,C 180,E1 -14128.814,E2 -14128.814} C_VEL
LIN {X 0,Y 339.209,Z 474.569,A -85,B 0,C 180,E1 -14131.188,E2 -14131.188} C_VEL
LIN {X 0,Y 339.108,Z 473.351,A -85,B 0,C 180,E1 -14133.565,E2 -14133.565} C_VEL
LIN {X 0,Y 339.247,Z 470.807,A -85,B 0,C 180,E1 -14136.067,E2 -14136.067} C_VEL
LIN {X 0,Y 339.444,Z 466.234,A -85,B 0,C 180,E1 -14138.934,E2 -14138.934} C_VEL
LIN {X 0,Y 339.918,Z 460.91,A -85,B 0,C 180,E1 -14141.328,E2 -14141.328} C_VEL
LIN {X 0,Y 340.722,Z 454.113,A -85,B 0,C 180,E1 -14143.723,E2 -14143.723} C_VEL
LIN {X 0,Y 341.976,Z 445.664,A -85,B 0,C 180,E1 -14146.108,E2 -14146.108} C_VEL
LIN {X 0,Y 343.436,Z 436.65,A -85,B 0,C 180,E1 -14148.185,E2 -14148.185} C_VEL
LIN {X 0,Y 344.997,Z 427.466,A -85,B 0,C 180,E1 -14149.952,E2 -14149.952} C_VEL
LIN {X 0,Y 346.766,Z 416.648,A -85,B 0,C 180,E1 -14151.709,E2 -14151.709} C_VEL
LIN {X 0,Y 348.739,Z 404.885,A -85,B 0,C 180,E1 -14153.298,E2 -14153.298} C_VEL
LIN {X 0,Y 350.697,Z 392.069,A -85,B 0,C 180,E1 -14154.73,E2 -14154.73} C_VEL
LIN {X 0,Y 352.824,Z 378.02,A -85,B 0,C 180,E1 -14155.991,E2 -14155.991} C_VEL
LIN {X 0,Y 353.427,Z 373.358,A -85,B 0,C 180,E1 -14156.36,E2 -14156.36} C_VEL
LIN {X 0,Y 351.437,Z 359.128,A -85,B 0,C 180,E1 -14157.572,E2 -14157.572} C_VEL
LIN {X 0,Y 348.589,Z 344.037,A -85,B 0,C 180,E1 -14158.678,E2 -14158.678} C_VEL
LIN {X 0,Y 344.805,Z 329.109,A -85,B 0,C 180,E1 -14159.629,E2 -14159.629} C_VEL
LIN {X 0,Y 341.536,Z 317.746,A -85,B 0,C 180,E1 -14160.246,E2 -14160.246} C_VEL
LIN {X 0,Y 341.513,Z 317.266,A -85,B 0,C 180,E1 -14160.297,E2 -14160.297} C_VEL
LIN {X 0,Y 342.089,Z 311.182,A -85,B 0,C 180,E1 -14163.691,E2 -14163.691} C_VEL
LIN {X 0,Y 342.781,Z 305.556,A -85,B 0,C 180,E1 -14166.906,E2 -14166.906} C_VEL
LIN {X 0,Y 343.485,Z 300.174,A -85,B 0,C 180,E1 -14170.098,E2 -14170.098} C_VEL
LIN {X 0,Y 343.766,Z 296.134,A -85,B 0,C 180,E1 -14172.608,E2 -14172.608} C_VEL
LIN {X 0,Y 343.364,Z 292.414,A -85,B 0,C 180,E1 -14175.077,E2 -14175.077} C_VEL
LIN {X 0,Y 342.369,Z 286.999,A -85,B 0,C 180,E1 -14178.936,E2 -14178.936} C_VEL
LIN {X 0,Y 341.666,Z 283.129,A -85,B 0,C 180,E1 -14181.895,E2 -14181.895} C_VEL
LIN {X 0,Y 340.933,Z 278.629,A -85,B 0,C 180,E1 -14185.545,E2 -14185.545} C_VEL
LIN {X 0,Y 340.725,Z 277.669,A -85,B 0,C 180,E1 -14186.511,E2 -14186.511} C_VEL
LIN {X 0,Y 340.748,Z 277.665,A -85,B 0,C 180,E1 -14190.329,E2 -14190.329} C_VEL
LIN {X 0,Y 340.809,Z 277.659,A -85,B 0,C 180,E1 -14193.019,E2 -14193.019} C_VEL
LIN {X 0,Y 340.762,Z 277.661,A -85,B 0,C 180,E1 -14195.638,E2 -14195.638} C_VEL
LIN {X 0,Y 340.759,Z 277.661,A -85,B 0,C 180,E1 -14199.474,E2 -14199.474} C_VEL
LIN {X 0,Y 340.864,Z 277.648,A -85,B 0,C 180,E1 -14201.983,E2 -14201.983} C_VEL
LIN {X 0,Y 340.875,Z 277.646,A -85,B 0,C 180,E1 -14205.704,E2 -14205.704} C_VEL
LIN {X 0,Y 340.876,Z 277.647,A -85,B 0,C 180,E1 -14209.305,E2 -14209.305} C_VEL
LIN {X 0,Y 341.021,Z 277.63,A -85,B 0,C 180,E1 -14212.896,E2 -14212.896} C_VEL
LIN {X 0,Y 341.172,Z 277.609,A -85,B 0,C 180,E1 -14217.638,E2 -14217.638} C_VEL
LIN {X 0,Y 341.301,Z 277.595,A -85,B 0,C 180,E1 -14219.999,E2 -14219.999} C_VEL
LIN {X 0,Y 341.171,Z 277.614,A -85,B 0,C 180,E1 -14222.36,E2 -14222.36} C_VEL
LIN {X 0,Y 341.079,Z 277.621,A -85,B 0,C 180,E1 -14227.1,E2 -14227.1} C_VEL
LIN {X 0,Y 340.874,Z 277.647,A -85,B 0,C 180,E1 -14230.692,E2 -14230.692} C_VEL
LIN {X 0,Y 340.865,Z 277.652,A -85,B 0,C 180,E1 -14234.323,E2 -14234.323} C_VEL
LIN {X 0,Y 340.839,Z 277.652,A -85,B 0,C 180,E1 -14238.465,E2 -14238.465} C_VEL
LIN {X 0,Y 340.754,Z 277.662,A -85,B 0,C 180,E1 -14241.855,E2 -14241.855} C_VEL
LIN {X 0,Y 340.772,Z 277.661,A -85,B 0,C 180,E1 -14245.663,E2 -14245.663} C_VEL
LIN {X 0,Y 340.727,Z 277.666,A -85,B 0,C 180,E1 -14248.319,E2 -14248.319} C_VEL
LIN {X 0,Y 340.696,Z 277.668,A -85,B 0,C 180,E1 -14251.043,E2 -14251.043} C_VEL
LIN {X 0,Y 340.716,Z 277.665,A -85,B 0,C 180,E1 -14255.277,E2 -14255.277} C_VEL
LIN {X 0,Y 340.707,Z 277.668,A -85,B 0,C 180,E1 -14258.384,E2 -14258.384} C_VEL
LIN {X 0,Y 340.698,Z 277.67,A -85,B 0,C 180,E1 -14262.044,E2 -14262.044} C_VEL
LIN {X 0,Y 340.733,Z 277.666,A -85,B 0,C 180,E1 -14265.469,E2 -14265.469} C_VEL
LIN {X 0,Y 340.722,Z 277.664,A -85,B 0,C 180,E1 -14268.695,E2 -14268.695} C_VEL
LIN {X 0,Y 340.733,Z 277.67,A -85,B 0,C 180,E1 -14271.772,E2 -14271.772} C_VEL
LIN {X 0,Y 340.716,Z 277.669,A -85,B 0,C 180,E1 -14275.594,E2 -14275.594} C_VEL
LIN {X 0,Y 340.697,Z 277.669,A -85,B 0,C 180,E1 -14278.954,E2 -14278.954} C_VEL
LIN {X 0,Y 340.772,Z 277.659,A -85,B 0,C 180,E1 -14282.472,E2 -14282.472} C_VEL
LIN {X 0,Y 340.748,Z 277.668,A -85,B 0,C 180,E1 -14285.637,E2 -14285.637} C_VEL
LIN {X 0,Y 340.74,Z 277.668,A -85,B 0,C 180,E1 -14289.473,E2 -14289.473} C_VEL
LIN {X 0,Y 340.849,Z 277.65,A -85,B 0,C 180,E1 -14291.983,E2 -14291.983} C_VEL
LIN {X 0,Y 340.86,Z 277.651,A -85,B 0,C 180,E1 -14295.704,E2 -14295.704} C_VEL
LIN {X 0,Y 340.865,Z 277.652,A -85,B 0,C 180,E1 -14299.305,E2 -14299.305} C_VEL
LIN {X 0,Y 341.063,Z 277.622,A -85,B 0,C 180,E1 -14302.897,E2 -14302.897} C_VEL
LIN {X 0,Y 341.021,Z 277.629,A -85,B 0,C 180,E1 -14304.085,E2 -14304.085} C_VEL
LIN {X 0,Y 340.579,Z 277.688,A -85,B 0,C 180,E1 -14307.634,E2 -14307.634} C_VEL
LIN {X 0,Y 340.939,Z 277.968,A -85,B 0,C 180,E1 -14308.818,E2 -14308.818} C_VEL
LIN {X 0,Y 340.176,Z 281.285,A -85,B 0,C 180,E1 -14312.96,E2 -14312.96} C_VEL
LIN {X 0,Y 341.272,Z 284.369,A -85,B 0,C 180,E1 -14313.151,E2 -14313.151} C_VEL
LIN {X 0,Y 345.592,Z 294.511,A -85,B 0,C 180,E1 -14313.887,E2 -14313.887} C_VEL
LIN {X 0,Y 350.405,Z 308.19,A -85,B 0,C 180,E1 -14314.957,E2 -14314.957} C_VEL
LIN {X 0,Y 354.238,Z 321.606,A -85,B 0,C 180,E1 -14316.12,E2 -14316.12} C_VEL
LIN {X 0,Y 354.974,Z 324.603,A -85,B 0,C 180,E1 -14316.393,E2 -14316.393} C_VEL
LIN {X 0,Y 353.404,Z 338.682,A -85,B 0,C 180,E1 -14317.448,E2 -14317.448} C_VEL
LIN {X 0,Y 351.607,Z 352.71,A -85,B 0,C 180,E1 -14318.766,E2 -14318.766} C_VEL
LIN {X 0,Y 349.857,Z 364.876,A -85,B 0,C 180,E1 -14320.17,E2 -14320.17} C_VEL
LIN {X 0,Y 348.038,Z 376.583,A -85,B 0,C 180,E1 -14321.797,E2 -14321.797} C_VEL
LIN {X 0,Y 346.147,Z 387.441,A -85,B 0,C 180,E1 -14323.603,E2 -14323.603} C_VEL
LIN {X 0,Y 344.618,Z 396.339,A -85,B 0,C 180,E1 -14325.373,E2 -14325.373} C_VEL
LIN {X 0,Y 343.021,Z 405.606,A -85,B 0,C 180,E1 -14327.589,E2 -14327.589} C_VEL
LIN {X 0,Y 341.794,Z 413.236,A -85,B 0,C 180,E1 -14329.832,E2 -14329.832} C_VEL
LIN {X 0,Y 340.888,Z 419.03,A -85,B 0,C 180,E1 -14331.918,E2 -14331.918} C_VEL
LIN {X 0,Y 340.082,Z 424.467,A -85,B 0,C 180,E1 -14334.412,E2 -14334.412} C_VEL
LIN {X 0,Y 339.789,Z 426.76,A -85,B 0,C 180,E1 -14335.743,E2 -14335.743} C_VEL
LIN {X 0,Y 339.529,Z 428.725,A -85,B 0,C 180,E1 -14337.122,E2 -14337.122} C_VEL
LIN {X 0,Y 339.164,Z 431.418,A -85,B 0,C 180,E1 -14339.822,E2 -14339.822} C_VEL
LIN {X 0,Y 339.104,Z 432.487,A -85,B 0,C 180,E1 -14341.821,E2 -14341.821} C_VEL
LIN {X 0,Y 339.069,Z 432.671,A -85,B 0,C 180,E1 -14344.03,E2 -14344.03} C_VEL
LIN {X 0,Y 339.191,Z 432.009,A -85,B 0,C 180,E1 -14346.095,E2 -14346.095} C_VEL
LIN {X 0,Y 339.474,Z 430.254,A -85,B 0,C 180,E1 -14348.394,E2 -14348.394} C_VEL
LIN {X 0,Y 339.807,Z 428.251,A -85,B 0,C 180,E1 -14350.074,E2 -14350.074} C_VEL
LIN {X 0,Y 340.305,Z 425.261,A -85,B 0,C 180,E1 -14351.975,E2 -14351.975} C_VEL
LIN {X 0,Y 341.154,Z 420.117,A -85,B 0,C 180,E1 -14354.46,E2 -14354.46} C_VEL
LIN {X 0,Y 342.25,Z 414.1,A -85,B 0,C 180,E1 -14356.709,E2 -14356.709} C_VEL
LIN {X 0,Y 343.56,Z 407.404,A -85,B 0,C 180,E1 -14358.743,E2 -14358.743} C_VEL
LIN {X 0,Y 345.19,Z 398.922,A -85,B 0,C 180,E1 -14360.867,E2 -14360.867} C_VEL
LIN {X 0,Y 345.791,Z 395.621,A -85,B 0,C 180,E1 -14361.597,E2 -14361.597} C_VEL
LIN {X 0,Y 345.8,Z 392.082,A -85,B 0,C 180,E1 -14362.375,E2 -14362.375} C_VEL
LIN {X 0,Y 343.008,Z 381.341,A -85,B 0,C 180,E1 -14364.703,E2 -14364.703} C_VEL
LIN {X 0,Y 342.893,Z 377.271,A -85,B 0,C 180,E1 -14365.423,E2 -14365.423} C_VEL
LIN {X 0,Y 343.117,Z 375.83,A -85,B 0,C 180,E1 -14365.648,E2 -14365.648} C_VEL
LIN {X 0,Y 345.396,Z 363.385,A -85,B 0,C 180,E1 -14367.338,E2 -14367.338} C_VEL
LIN {X 0,Y 347.378,Z 350.901,A -85,B 0,C 180,E1 -14368.734,E2 -14368.734} C_VEL
LIN {X 0,Y 349.272,Z 337.963,A -85,B 0,C 180,E1 -14369.908,E2 -14369.908} C_VEL
LIN {X 0,Y 350.268,Z 328.676,A -85,B 0,C 180,E1 -14370.635,E2 -14370.635} C_VEL
LIN {X 0,Y 347.46,Z 318.375,A -85,B 0,C 180,E1 -14371.683,E2 -14371.683} C_VEL
LIN {X 0,Y 342.923,Z 305.559,A -85,B 0,C 180,E1 -14372.955,E2 -14372.955} C_VEL
LIN {X 0,Y 337.213,Z 292.338,A -85,B 0,C 180,E1 -14374.21,E2 -14374.21} C_VEL
LIN {X 0,Y 333.861,Z 285.826,A -85,B 0,C 180,E1 -14374.832,E2 -14374.832} C_VEL
LIN {X 0,Y 333.642,Z 284.725,A -85,B 0,C 180,E1 -14374.925,E2 -14374.925} C_VEL
LIN {X 0,Y 333.831,Z 282.154,A -85,B 0,C 180,E1 -14379.031,E2 -14379.031} C_VEL
LIN {X 0,Y 333.923,Z 280.622,A -85,B 0,C 180,E1 -14381.598,E2 -14381.598} C_VEL
LIN {X 0,Y 333.8,Z 278.533,A -85,B 0,C 180,E1 -14385.579,E2 -14385.579} C_VEL
LIN {X 0,Y 333.827,Z 278.53,A -85,B 0,C 180,E1 -14389.079,E2 -14389.079} C_VEL
LIN {X 0,Y 334.02,Z 278.503,A -85,B 0,C 180,E1 -14392.749,E2 -14392.749} C_VEL
LIN {X 0,Y 333.808,Z 278.532,A -85,B 0,C 180,E1 -14395.17,E2 -14395.17} C_VEL
LIN {X 0,Y 334.103,Z 278.492,A -85,B 0,C 180,E1 -14397.59,E2 -14397.59} C_VEL
LIN {X 0,Y 334.243,Z 278.473,A -85,B 0,C 180,E1 -14400.001,E2 -14400.001} C_VEL
LIN {X 0,Y 334.103,Z 278.491,A -85,B 0,C 180,E1 -14402.412,E2 -14402.412} C_VEL
LIN {X 0,Y 334.022,Z 278.505,A -85,B 0,C 180,E1 -14407.254,E2 -14407.254} C_VEL
LIN {X 0,Y 333.83,Z 278.523,A -85,B 0,C 180,E1 -14410.923,E2 -14410.923} C_VEL
LIN {X 0,Y 333.805,Z 278.527,A -85,B 0,C 180,E1 -14414.636,E2 -14414.636} C_VEL
LIN {X 0,Y 333.794,Z 278.531,A -85,B 0,C 180,E1 -14418.657,E2 -14418.657} C_VEL
LIN {X 0,Y 333.69,Z 278.546,A -85,B 0,C 180,E1 -14422.279,E2 -14422.279} C_VEL
LIN {X 0,Y 333.734,Z 278.542,A -85,B 0,C 180,E1 -14426.248,E2 -14426.248} C_VEL
LIN {X 0,Y 333.709,Z 278.544,A -85,B 0,C 180,E1 -14428.973,E2 -14428.973} C_VEL
LIN {X 0,Y 333.767,Z 279.043,A -85,B 0,C 180,E1 -14430.356,E2 -14430.356} C_VEL
LIN {X 0,Y 334.424,Z 282.572,A -85,B 0,C 180,E1 -14434.571,E2 -14434.571} C_VEL
LIN {X 0,Y 334.873,Z 285.408,A -85,B 0,C 180,E1 -14437.491,E2 -14437.491} C_VEL
LIN {X 0,Y 335.542,Z 289.319,A -85,B 0,C 180,E1 -14441.061,E2 -14441.061} C_VEL
LIN {X 0,Y 336.336,Z 293.819,A -85,B 0,C 180,E1 -14444.729,E2 -14444.729} C_VEL
LIN {X 0,Y 336.773,Z 296.729,A -85,B 0,C 180,E1 -14446.921,E2 -14446.921} C_VEL
LIN {X 0,Y 336.668,Z 299.357,A -85,B 0,C 180,E1 -14448.722,E2 -14448.722} C_VEL
LIN {X 0,Y 335.764,Z 305.461,A -85,B 0,C 180,E1 -14452.628,E2 -14452.628} C_VEL
LIN {X 0,Y 335.021,Z 311.419,A -85,B 0,C 180,E1 -14456.228,E2 -14456.228} C_VEL
LIN {X 0,Y 334.639,Z 314.996,A -85,B 0,C 180,E1 -14458.202,E2 -14458.202} C_VEL
LIN {X 0,Y 335.635,Z 318.314,A -85,B 0,C 180,E1 -14458.415,E2 -14458.415} C_VEL
LIN {X 0,Y 340.267,Z 332.514,A -85,B 0,C 180,E1 -14459.447,E2 -14459.447} C_VEL
LIN {X 0,Y 343.584,Z 346.467,A -85,B 0,C 180,E1 -14460.511,E2 -14460.511} C_VEL
LIN {X 0,Y 345.822,Z 360.28,A -85,B 0,C 180,E1 -14461.651,E2 -14461.651} C_VEL
LIN {X 0,Y 347.4,Z 373.674,A -85,B 0,C 180,E1 -14462.891,E2 -14462.891} C_VEL
LIN {X 0,Y 346.352,Z 382.393,A -85,B 0,C 180,E1 -14463.65,E2 -14463.65} C_VEL
LIN {X 0,Y 343.972,Z 396.551,A -85,B 0,C 180,E1 -14465.077,E2 -14465.077} C_VEL
LIN {X 0,Y 341.642,Z 409.382,A -85,B 0,C 180,E1 -14466.673,E2 -14466.673} C_VEL
LIN {X 0,Y 339.574,Z 420.806,A -85,B 0,C 180,E1 -14468.398,E2 -14468.398} C_VEL
LIN {X 0,Y 337.782,Z 430.998,A -85,B 0,C 180,E1 -14470.24,E2 -14470.24} C_VEL
LIN {X 0,Y 335.932,Z 440.757,A -85,B 0,C 180,E1 -14472.342,E2 -14472.342} C_VEL
LIN {X 0,Y 334.552,Z 448.943,A -85,B 0,C 180,E1 -14474.465,E2 -14474.465} C_VEL
LIN {X 0,Y 333.474,Z 455.769,A -85,B 0,C 180,E1 -14476.596,E2 -14476.596} C_VEL
LIN {X 0,Y 332.688,Z 462.069,A -85,B 0,C 180,E1 -14479.041,E2 -14479.041} C_VEL
LIN {X 0,Y 332.297,Z 466.961,A -85,B 0,C 180,E1 -14481.487,E2 -14481.487} C_VEL
LIN {X 0,Y 332.144,Z 470.636,A -85,B 0,C 180,E1 -14483.992,E2 -14483.992} C_VEL
LIN {X 0,Y 332.042,Z 472.921,A -85,B 0,C 180,E1 -14486.36,E2 -14486.36} C_VEL
LIN {X 0,Y 332.119,Z 474.113,A -85,B 0,C 180,E1 -14488.788,E2 -14488.788} C_VEL
LIN {X 0,Y 332.118,Z 474.128,A -85,B 0,C 180,E1 -14491.213,E2 -14491.213} C_VEL
LIN {X 0,Y 332.035,Z 472.903,A -85,B 0,C 180,E1 -14493.642,E2 -14493.642} C_VEL
LIN {X 0,Y 332.151,Z 470.496,A -85,B 0,C 180,E1 -14496.074,E2 -14496.074} C_VEL
LIN {X 0,Y 332.308,Z 466.844,A -85,B 0,C 180,E1 -14498.514,E2 -14498.514} C_VEL
LIN {X 0,Y 332.689,Z 461.864,A -85,B 0,C 180,E1 -14500.961,E2 -14500.961} C_VEL
LIN {X 0,Y 333.506,Z 455.439,A -85,B 0,C 180,E1 -14503.404,E2 -14503.404} C_VEL
LIN {X 0,Y 334.698,Z 447.385,A -85,B 0,C 180,E1 -14505.842,E2 -14505.842} C_VEL
LIN {X 0,Y 336.077,Z 438.809,A -85,B 0,C 180,E1 -14507.967,E2 -14507.967} C_VEL
LIN {X 0,Y 337.748,Z 430.143,A -85,B 0,C 180,E1 -14509.764,E2 -14509.764} C_VEL
LIN {X 0,Y 339.45,Z 419.61,A -85,B 0,C 180,E1 -14511.606,E2 -14511.606} C_VEL
LIN {X 0,Y 341.544,Z 407.671,A -85,B 0,C 180,E1 -14513.336,E2 -14513.336} C_VEL
LIN {X 0,Y 343.521,Z 395.475,A -85,B 0,C 180,E1 -14514.798,E2 -14514.798} C_VEL
LIN {X 0,Y 345.693,Z 382.289,A -85,B 0,C 180,E1 -14516.082,E2 -14516.082} C_VEL
LIN {X 0,Y 346.79,Z 374.262,A -85,B 0,C 180,E1 -14516.751,E2 -14516.751} C_VEL
LIN {X 0,Y 344.756,Z 359.696,A -85,B 0,C 180,E1 -14518.044,E2 -14518.044} C_VEL
LIN {X 0,Y 342.102,Z 345.52,A -85,B 0,C 180,E1 -14519.13,E2 -14519.13} C_VEL
LIN {X 0,Y 338.596,Z 331.341,A -85,B 0,C 180,E1 -14520.08,E2 -14520.08} C_VEL
LIN {X 0,Y 334.574,Z 316.914,A -85,B 0,C 180,E1 -14520.92,E2 -14520.92} C_VEL
LIN {X 0,Y 335.197,Z 310.686,A -85,B 0,C 180,E1 -14524.48,E2 -14524.48} C_VEL
LIN {X 0,Y 336.014,Z 304.53,A -85,B 0,C 180,E1 -14528.099,E2 -14528.099} C_VEL
LIN {X 0,Y 336.664,Z 299.384,A -85,B 0,C 180,E1 -14531.277,E2 -14531.277} C_VEL
LIN {X 0,Y 336.691,Z 295.888,A -85,B 0,C 180,E1 -14533.539,E2 -14533.539} C_VEL
LIN {X 0,Y 336.012,Z 291.859,A -85,B 0,C 180,E1 -14536.351,E2 -14536.351} C_VEL
LIN {X 0,Y 335.252,Z 287.652,A -85,B 0,C 180,E1 -14539.468,E2 -14539.468} C_VEL
LIN {X 0,Y 334.493,Z 283.201,A -85,B 0,C 180,E1 -14542.98,E2 -14542.98} C_VEL
LIN {X 0,Y 334.021,Z 280.308,A -85,B 0,C 180,E1 -14545.381,E2 -14545.381} C_VEL
LIN {X 0,Y 333.675,Z 278.547,A -85,B 0,C 180,E1 -14546.978,E2 -14546.978} C_VEL
LIN {X 0,Y 333.696,Z 278.546,A -85,B 0,C 180,E1 -14551.025,E2 -14551.025} C_VEL
LIN {X 0,Y 333.741,Z 278.536,A -85,B 0,C 180,E1 -14553.753,E2 -14553.753} C_VEL
LIN {X 0,Y 333.726,Z 278.538,A -85,B 0,C 180,E1 -14557.913,E2 -14557.913} C_VEL
LIN {X 0,Y 333.8,Z 278.528,A -85,B 0,C 180,E1 -14561.589,E2 -14561.589} C_VEL
LIN {X 0,Y 333.814,Z 278.526,A -85,B 0,C 180,E1 -14565.576,E2 -14565.576} C_VEL
LIN {X 0,Y 333.839,Z 278.525,A -85,B 0,C 180,E1 -14569.077,E2 -14569.077} C_VEL
LIN {X 0,Y 333.973,Z 278.51,A -85,B 0,C 180,E1 -14572.745,E2 -14572.745} C_VEL
LIN {X 0,Y 333.808,Z 278.527,A -85,B 0,C 180,E1 -14575.168,E2 -14575.168} C_VEL
LIN {X 0,Y 334.11,Z 278.489,A -85,B 0,C 180,E1 -14577.588,E2 -14577.588} C_VEL
LIN {X 0,Y 334.252,Z 278.473,A -85,B 0,C 180,E1 -14579.999,E2 -14579.999} C_VEL
LIN {X 0,Y 334.108,Z 278.493,A -85,B 0,C 180,E1 -14582.41,E2 -14582.41} C_VEL
LIN {X 0,Y 334.029,Z 278.499,A -85,B 0,C 180,E1 -14587.251,E2 -14587.251} C_VEL
LIN {X 0,Y 333.837,Z 278.521,A -85,B 0,C 180,E1 -14590.92,E2 -14590.92} C_VEL
LIN {X 0,Y 333.811,Z 278.528,A -85,B 0,C 180,E1 -14594.633,E2 -14594.633} C_VEL
LIN {X 0,Y 333.798,Z 278.527,A -85,B 0,C 180,E1 -14598.654,E2 -14598.654} C_VEL
LIN {X 0,Y 333.693,Z 278.545,A -85,B 0,C 180,E1 -14602.276,E2 -14602.276} C_VEL
LIN {X 0,Y 333.735,Z 278.538,A -85,B 0,C 180,E1 -14606.245,E2 -14606.245} C_VEL
LIN {X 0,Y 333.689,Z 278.539,A -85,B 0,C 180,E1 -14608.972,E2 -14608.972} C_VEL
LIN {X 0,Y 333.644,Z 278.548,A -85,B 0,C 180,E1 -14612.586,E2 -14612.586} C_VEL
LIN {X 0,Y 333.674,Z 278.545,A -85,B 0,C 180,E1 -14616.137,E2 -14616.137} C_VEL
LIN {X 0,Y 333.644,Z 278.547,A -85,B 0,C 180,E1 -14619.19,E2 -14619.19} C_VEL
LIN {X 0,Y 333.637,Z 278.545,A -85,B 0,C 180,E1 -14622.5,E2 -14622.5} C_VEL
LIN {X 0,Y 333.681,Z 278.547,A -85,B 0,C 180,E1 -14625.968,E2 -14625.968} C_VEL
LIN {X 0,Y 333.697,Z 278.54,A -85,B 0,C 180,E1 -14629.303,E2 -14629.303} C_VEL
LIN {X 0,Y 333.66,Z 278.546,A -85,B 0,C 180,E1 -14633.166,E2 -14633.166} C_VEL
LIN {X 0,Y 333.668,Z 278.545,A -85,B 0,C 180,E1 -14635.34,E2 -14635.34} C_VEL
LIN {X 0,Y 333.696,Z 278.544,A -85,B 0,C 180,E1 -14639.709,E2 -14639.709} C_VEL
LIN {X 0,Y 333.737,Z 278.536,A -85,B 0,C 180,E1 -14642.4,E2 -14642.4} C_VEL
LIN {X 0,Y 333.719,Z 278.539,A -85,B 0,C 180,E1 -14645.089,E2 -14645.089} C_VEL
LIN {X 0,Y 333.673,Z 278.544,A -85,B 0,C 180,E1 -14649.018,E2 -14649.018} C_VEL
LIN {X 0,Y 333.786,Z 278.533,A -85,B 0,C 180,E1 -14651.588,E2 -14651.588} C_VEL
LIN {X 0,Y 333.799,Z 278.532,A -85,B 0,C 180,E1 -14655.575,E2 -14655.575} C_VEL
LIN {X 0,Y 333.828,Z 278.526,A -85,B 0,C 180,E1 -14659.077,E2 -14659.077} C_VEL
LIN {X 0,Y 334.013,Z 278.498,A -85,B 0,C 180,E1 -14662.746,E2 -14662.746} C_VEL
LIN {X 0,Y 334,Z 278.504,A -85,B 0,C 180,E1 -14663.96,E2 -14663.96} C_VEL
LIN {X 0,Y 333.528,Z 278.567,A -85,B 0,C 180,E1 -14667.584,E2 -14667.584} C_VEL
LIN {X 0,Y 333.9,Z 278.915,A -85,B 0,C 180,E1 -14668.793,E2 -14668.793} C_VEL
LIN {X 0,Y 333.101,Z 281.668,A -85,B 0,C 180,E1 -14672.304,E2 -14672.304} C_VEL
LIN {X 0,Y 334.225,Z 284.811,A -85,B 0,C 180,E1 -14672.508,E2 -14672.508} C_VEL
LIN {X 0,Y 339.686,Z 297.615,A -85,B 0,C 180,E1 -14673.487,E2 -14673.487} C_VEL
LIN {X 0,Y 344.241,Z 310.824,A -85,B 0,C 180,E1 -14674.573,E2 -14674.573} C_VEL
LIN {X 0,Y 348.243,Z 325.267,A -85,B 0,C 180,E1 -14675.893,E2 -14675.893} C_VEL
LIN {X 0,Y 348.293,Z 327.585,A -85,B 0,C 180,E1 -14676.08,E2 -14676.08} C_VEL
LIN {X 0,Y 346.727,Z 340.919,A -85,B 0,C 180,E1 -14677.131,E2 -14677.131} C_VEL
LIN {X 0,Y 344.807,Z 354.825,A -85,B 0,C 180,E1 -14678.497,E2 -14678.497} C_VEL
LIN {X 0,Y 342.942,Z 367.388,A -85,B 0,C 180,E1 -14680.016,E2 -14680.016} C_VEL
LIN {X 0,Y 341.162,Z 378.237,A -85,B 0,C 180,E1 -14681.586,E2 -14681.586} C_VEL
LIN {X 0,Y 339.232,Z 388.995,A -85,B 0,C 180,E1 -14683.446,E2 -14683.446} C_VEL
LIN {X 0,Y 337.512,Z 398.366,A -85,B 0,C 180,E1 -14685.395,E2 -14685.395} C_VEL
LIN {X 0,Y 336.099,Z 406.161,A -85,B 0,C 180,E1 -14687.335,E2 -14687.335} C_VEL
LIN {X 0,Y 334.826,Z 413.768,A -85,B 0,C 180,E1 -14689.623,E2 -14689.623} C_VEL
LIN {X 0,Y 333.738,Z 420.363,A -85,B 0,C 180,E1 -14692.099,E2 -14692.099} C_VEL
LIN {X 0,Y 333.065,Z 424.812,A -85,B 0,C 180,E1 -14694.213,E2 -14694.213} C_VEL
LIN {X 0,Y 332.569,Z 428.275,A -85,B 0,C 180,E1 -14696.344,E2 -14696.344} C_VEL
LIN {X 0,Y 332.15,Z 431.379,A -85,B 0,C 180,E1 -14699.12,E2 -14699.12} C_VEL
LIN {X 0,Y 332.042,Z 432.367,A -85,B 0,C 180,E1 -14700.529,E2 -14700.529} C_VEL
LIN {X 0,Y 331.996,Z 433.003,A -85,B 0,C 180,E1 -14702.143,E2 -14702.143} C_VEL
LIN {X 0,Y 331.999,Z 433.092,A -85,B 0,C 180,E1 -14704.356,E2 -14704.356} C_VEL
LIN {X 0,Y 332.134,Z 432.279,A -85,B 0,C 180,E1 -14706.481,E2 -14706.481} C_VEL
LIN {X 0,Y 332.416,Z 430.707,A -85,B 0,C 180,E1 -14708.535,E2 -14708.535} C_VEL
LIN {X 0,Y 332.924,Z 427.828,A -85,B 0,C 180,E1 -14710.873,E2 -14710.873} C_VEL
LIN {X 0,Y 333.638,Z 423.837,A -85,B 0,C 180,E1 -14713.202,E2 -14713.202} C_VEL
LIN {X 0,Y 334.587,Z 418.528,A -85,B 0,C 180,E1 -14715.574,E2 -14715.574} C_VEL
LIN {X 0,Y 335.954,Z 411.658,A -85,B 0,C 180,E1 -14717.98,E2 -14717.98} C_VEL
LIN {X 0,Y 337.414,Z 404.585,A -85,B 0,C 180,E1 -14719.999,E2 -14719.999} C_VEL
LIN {X 0,Y 339.062,Z 396.311,A -85,B 0,C 180,E1 -14721.965,E2 -14721.965} C_VEL
LIN {X 0,Y 341.157,Z 386.177,A -85,B 0,C 180,E1 -14723.955,E2 -14723.955} C_VEL
LIN {X 0,Y 343.117,Z 375.83,A -85,B 0,C 180,E1 -14725.648,E2 -14725.648} C_VEL
LIN {X 0,Y 343.364,Z 371.555,A -85,B 0,C 180,E1 -14726.329,E2 -14726.329} C_VEL
LIN {X 0,Y 342.009,Z 364.594,A -85,B 0,C 180,E1 -14727.493,E2 -14727.493} C_VEL
LIN {X 0,Y 340.671,Z 357.32,A -85,B 0,C 180,E1 -14728.596,E2 -14728.596} C_VEL
LIN {X 0,Y 340.916,Z 352.485,A -85,B 0,C 180,E1 -14729.169,E2 -14729.169} C_VEL
LIN {X 0,Y 342.884,Z 339.62,A -85,B 0,C 180,E1 -14730.38,E2 -14730.38} C_VEL
LIN {X 0,Y 343.973,Z 331.602,A -85,B 0,C 180,E1 -14731.016,E2 -14731.016} C_VEL
LIN {X 0,Y 343.494,Z 328.345,A -85,B 0,C 180,E1 -14731.349,E2 -14731.349} C_VEL
LIN {X 0,Y 339.691,Z 315.508,A -85,B 0,C 180,E1 -14732.718,E2 -14732.718} C_VEL
LIN {X 0,Y 334.592,Z 302.235,A -85,B 0,C 180,E1 -14734.076,E2 -14734.076} C_VEL
LIN {X 0,Y 329.877,Z 292.285,A -85,B 0,C 180,E1 -14735.1,E2 -14735.1} C_VEL
LIN {X 0,Y 327.784,Z 288.408,A -85,B 0,C 180,E1 -14735.498,E2 -14735.498} C_VEL
LIN {X 0,Y 326.641,Z 285.29,A -85,B 0,C 180,E1 -14735.788,E2 -14735.788} C_VEL
LIN {X 0,Y 326.786,Z 283.59,A -85,B 0,C 180,E1 -14738.557,E2 -14738.557} C_VEL
LIN {X 0,Y 326.897,Z 282.063,A -85,B 0,C 180,E1 -14741.188,E2 -14741.188} C_VEL
LIN {X 0,Y 326.827,Z 279.975,A -85,B 0,C 180,E1 -14745.047,E2 -14745.047} C_VEL
LIN {X 0,Y 326.749,Z 279.41,A -85,B 0,C 180,E1 -14746.316,E2 -14746.316} C_VEL
LIN {X 0,Y 326.808,Z 279.404,A -85,B 0,C 180,E1 -14750.095,E2 -14750.095} C_VEL
LIN {X 0,Y 326.974,Z 279.38,A -85,B 0,C 180,E1 -14752.592,E2 -14752.592} C_VEL
LIN {X 0,Y 326.775,Z 279.408,A -85,B 0,C 180,E1 -14755.066,E2 -14755.066} C_VEL
LIN {X 0,Y 327.043,Z 279.371,A -85,B 0,C 180,E1 -14757.538,E2 -14757.538} C_VEL
LIN {X 0,Y 327.194,Z 279.351,A -85,B 0,C 180,E1 -14760.001,E2 -14760.001} C_VEL
LIN {X 0,Y 327.044,Z 279.371,A -85,B 0,C 180,E1 -14762.465,E2 -14762.465} C_VEL
LIN {X 0,Y 326.992,Z 279.376,A -85,B 0,C 180,E1 -14766.17,E2 -14766.17} C_VEL
LIN {X 0,Y 326.911,Z 279.386,A -85,B 0,C 180,E1 -14768.656,E2 -14768.656} C_VEL
LIN {X 0,Y 326.731,Z 279.409,A -85,B 0,C 180,E1 -14772.423,E2 -14772.423} C_VEL
LIN {X 0,Y 326.751,Z 279.404,A -85,B 0,C 180,E1 -14774.959,E2 -14774.959} C_VEL
LIN {X 0,Y 326.73,Z 279.409,A -85,B 0,C 180,E1 -14778.84,E2 -14778.84} C_VEL
LIN {X 0,Y 326.618,Z 279.426,A -85,B 0,C 180,E1 -14782.789,E2 -14782.789} C_VEL
LIN {X 0,Y 326.688,Z 279.415,A -85,B 0,C 180,E1 -14785.485,E2 -14785.485} C_VEL
LIN {X 0,Y 326.654,Z 279.426,A -85,B 0,C 180,E1 -14788.252,E2 -14788.252} C_VEL
LIN {X 0,Y 326.92,Z 281.225,A -85,B 0,C 180,E1 -14791.062,E2 -14791.062} C_VEL
LIN {X 0,Y 327.356,Z 283.581,A -85,B 0,C 180,E1 -14793.932,E2 -14793.932} C_VEL
LIN {X 0,Y 327.962,Z 286.998,A -85,B 0,C 180,E1 -14797.546,E2 -14797.546} C_VEL
LIN {X 0,Y 328.676,Z 291.319,A -85,B 0,C 180,E1 -14801.55,E2 -14801.55} C_VEL
LIN {X 0,Y 329.482,Z 295.833,A -85,B 0,C 180,E1 -14805.26,E2 -14805.26} C_VEL
LIN {X 0,Y 329.791,Z 298.141,A -85,B 0,C 180,E1 -14807.006,E2 -14807.006} C_VEL
LIN {X 0,Y 329.479,Z 301.609,A -85,B 0,C 180,E1 -14809.416,E2 -14809.416} C_VEL
LIN {X 0,Y 328.641,Z 307.473,A -85,B 0,C 180,E1 -14813.219,E2 -14813.219} C_VEL
LIN {X 0,Y 327.722,Z 314.215,A -85,B 0,C 180,E1 -14817.332,E2 -14817.332} C_VEL
LIN {X 0,Y 328.748,Z 317.798,A -85,B 0,C 180,E1 -14817.582,E2 -14817.582} C_VEL
LIN {X 0,Y 333.342,Z 331.38,A -85,B 0,C 180,E1 -14818.637,E2 -14818.637} C_VEL
LIN {X 0,Y 336.894,Z 345.698,A -85,B 0,C 180,E1 -14819.786,E2 -14819.786} C_VEL
LIN {X 0,Y 339.263,Z 359.741,A -85,B 0,C 180,E1 -14820.988,E2 -14820.988} C_VEL
LIN {X 0,Y 340.88,Z 374.887,A -85,B 0,C 180,E1 -14822.443,E2 -14822.443} C_VEL
LIN {X 0,Y 340.433,Z 379.401,A -85,B 0,C 180,E1 -14822.845,E2 -14822.845} C_VEL
LIN {X 0,Y 338.248,Z 392.529,A -85,B 0,C 180,E1 -14824.131,E2 -14824.131} C_VEL
LIN {X 0,Y 335.953,Z 404.847,A -85,B 0,C 180,E1 -14825.597,E2 -14825.597} C_VEL
LIN {X 0,Y 333.543,Z 417.226,A -85,B 0,C 180,E1 -14827.386,E2 -14827.386} C_VEL
LIN {X 0,Y 331.568,Z 427.619,A -85,B 0,C 180,E1 -14829.205,E2 -14829.205} C_VEL
LIN {X 0,Y 329.848,Z 436.476,A -85,B 0,C 180,E1 -14831.04,E2 -14831.04} C_VEL
LIN {X 0,Y 328.213,Z 445.258,A -85,B 0,C 180,E1 -14833.198,E2 -14833.198} C_VEL
LIN {X 0,Y 326.749,Z 453.327,A -85,B 0,C 180,E1 -14835.61,E2 -14835.61} C_VEL
LIN {X 0,Y 325.884,Z 460.21,A -85,B 0,C 180,E1 -14838.179,E2 -14838.179} C_VEL
LIN {X 0,Y 325.281,Z 465.445,A -85,B 0,C 180,E1 -14840.675,E2 -14840.675} C_VEL
LIN {X 0,Y 325.11,Z 468.508,A -85,B 0,C 180,E1 -14842.548,E2 -14842.548} C_VEL
LIN {X 0,Y 324.99,Z 471.468,A -85,B 0,C 180,E1 -14845.039,E2 -14845.039} C_VEL
LIN {X 0,Y 324.96,Z 473.23,A -85,B 0,C 180,E1 -14847.522,E2 -14847.522} C_VEL
LIN {X 0,Y 325.08,Z 473.83,A -85,B 0,C 180,E1 -14850.001,E2 -14850.001} C_VEL
LIN {X 0,Y 324.956,Z 473.214,A -85,B 0,C 180,E1 -14852.48,E2 -14852.48} C_VEL
LIN {X 0,Y 325.007,Z 471.386,A -85,B 0,C 180,E1 -14854.963,E2 -14854.963} C_VEL
LIN {X 0,Y 325.097,Z 468.345,A -85,B 0,C 180,E1 -14857.454,E2 -14857.454} C_VEL
LIN {X 0,Y 325.392,Z 464.025,A -85,B 0,C 180,E1 -14859.951,E2 -14859.951} C_VEL
LIN {X 0,Y 326.091,Z 458.325,A -85,B 0,C 180,E1 -14862.447,E2 -14862.447} C_VEL
LIN {X 0,Y 327.075,Z 451.084,A -85,B 0,C 180,E1 -14864.943,E2 -14864.943} C_VEL
LIN {X 0,Y 328.364,Z 443.35,A -85,B 0,C 180,E1 -14867.116,E2 -14867.116} C_VEL
LIN {X 0,Y 330.107,Z 434.061,A -85,B 0,C 180,E1 -14869.269,E2 -14869.269} C_VEL
LIN {X 0,Y 331.797,Z 424.602,A -85,B 0,C 180,E1 -14871.106,E2 -14871.106} C_VEL
LIN {X 0,Y 334.017,Z 412.389,A -85,B 0,C 180,E1 -14873.073,E2 -14873.073} C_VEL
LIN {X 0,Y 336.203,Z 399.955,A -85,B 0,C 180,E1 -14874.714,E2 -14874.714} C_VEL
LIN {X 0,Y 338.284,Z 387.778,A -85,B 0,C 180,E1 -14876.031,E2 -14876.031} C_VEL
LIN {X 0,Y 340.132,Z 375.006,A -85,B 0,C 180,E1 -14877.171,E2 -14877.171} C_VEL
LIN {X 0,Y 338.194,Z 360.857,A -85,B 0,C 180,E1 -14878.477,E2 -14878.477} C_VEL
LIN {X 0,Y 335.447,Z 345.994,A -85,B 0,C 180,E1 -14879.662,E2 -14879.662} C_VEL
LIN {X 0,Y 331.822,Z 331.393,A -85,B 0,C 180,E1 -14880.687,E2 -14880.687} C_VEL
LIN {X 0,Y 327.593,Z 316.495,A -85,B 0,C 180,E1 -14881.585,E2 -14881.585} C_VEL
LIN {X 0,Y 328.405,Z 309.706,A -85,B 0,C 180,E1 -14885.587,E2 -14885.587} C_VEL
LIN {X 0,Y 329.179,Z 304.049,A -85,B 0,C 180,E1 -14889.038,E2 -14889.038} C_VEL
LIN {X 0,Y 329.696,Z 299.776,A -85,B 0,C 180,E1 -14891.747,E2 -14891.747} C_VEL
LIN {X 0,Y 329.718,Z 297.063,A -85,B 0,C 180,E1 -14893.554,E2 -14893.554} C_VEL
LIN {X 0,Y 328.924,Z 292.443,A -85,B 0,C 180,E1 -14896.863,E2 -14896.863} C_VEL
LIN {X 0,Y 328.024,Z 287.713,A -85,B 0,C 180,E1 -14900.473,E2 -14900.473} C_VEL
LIN {X 0,Y 327.524,Z 284.496,A -85,B 0,C 180,E1 -14903.07,E2 -14903.07} C_VEL
LIN {X 0,Y 326.93,Z 281.067,A -85,B 0,C 180,E1 -14906.018,E2 -14906.018} C_VEL
LIN {X 0,Y 326.612,Z 279.427,A -85,B 0,C 180,E1 -14907.638,E2 -14907.638} C_VEL
LIN {X 0,Y 326.654,Z 279.421,A -85,B 0,C 180,E1 -14910.339,E2 -14910.339} C_VEL
LIN {X 0,Y 326.696,Z 279.417,A -85,B 0,C 180,E1 -14914.516,E2 -14914.516} C_VEL
LIN {X 0,Y 326.655,Z 279.423,A -85,B 0,C 180,E1 -14918.545,E2 -14918.545} C_VEL
LIN {X 0,Y 326.751,Z 279.407,A -85,B 0,C 180,E1 -14921.177,E2 -14921.177} C_VEL
LIN {X 0,Y 326.769,Z 279.404,A -85,B 0,C 180,E1 -14925.432,E2 -14925.432} C_VEL
LIN {X 0,Y 326.775,Z 279.406,A -85,B 0,C 180,E1 -14928.838,E2 -14928.838} C_VEL
LIN {X 0,Y 326.928,Z 279.389,A -85,B 0,C 180,E1 -14932.588,E2 -14932.588} C_VEL
LIN {X 0,Y 326.774,Z 279.404,A -85,B 0,C 180,E1 -14935.064,E2 -14935.064} C_VEL
LIN {X 0,Y 327.05,Z 279.368,A -85,B 0,C 180,E1 -14937.535,E2 -14937.535} C_VEL
LIN {X 0,Y 327.203,Z 279.351,A -85,B 0,C 180,E1 -14939.999,E2 -14939.999} C_VEL
LIN {X 0,Y 327.049,Z 279.371,A -85,B 0,C 180,E1 -14942.462,E2 -14942.462} C_VEL
LIN {X 0,Y 326.974,Z 279.376,A -85,B 0,C 180,E1 -14946.675,E2 -14946.675} C_VEL
LIN {X 0,Y 326.817,Z 279.399,A -85,B 0,C 180,E1 -14949.905,E2 -14949.905} C_VEL
LIN {X 0,Y 326.761,Z 279.403,A -85,B 0,C 180,E1 -14953.684,E2 -14953.684} C_VEL
LIN {X 0,Y 326.701,Z 279.412,A -85,B 0,C 180,E1 -14957.526,E2 -14957.526} C_VEL
LIN {X 0,Y 326.666,Z 279.417,A -85,B 0,C 180,E1 -14960.133,E2 -14960.133} C_VEL
LIN {X 0,Y 326.652,Z 279.423,A -85,B 0,C 180,E1 -14964.127,E2 -14964.127} C_VEL
LIN {X 0,Y 326.682,Z 279.412,A -85,B 0,C 180,E1 -14966.856,E2 -14966.856} C_VEL
LIN {X 0,Y 326.633,Z 279.421,A -85,B 0,C 180,E1 -14970.608,E2 -14970.608} C_VEL
LIN {X 0,Y 326.606,Z 279.427,A -85,B 0,C 180,E1 -14974.017,E2 -14974.017} C_VEL
LIN {X 0,Y 326.625,Z 279.42,A -85,B 0,C 180,E1 -14977.237,E2 -14977.237} C_VEL
LIN {X 0,Y 326.576,Z 279.427,A -85,B 0,C 180,E1 -14981.13,E2 -14981.13} C_VEL
LIN {X 0,Y 326.59,Z 279.425,A -85,B 0,C 180,E1 -14984.753,E2 -14984.753} C_VEL
LIN {X 0,Y 326.618,Z 279.422,A -85,B 0,C 180,E1 -14988.16,E2 -14988.16} C_VEL
LIN {X 0,Y 326.641,Z 279.421,A -85,B 0,C 180,E1 -14991.393,E2 -14991.393} C_VEL
LIN {X 0,Y 326.613,Z 279.421,A -85,B 0,C 180,E1 -14994.85,E2 -14994.85} C_VEL
LIN {X 0,Y 326.601,Z 279.428,A -85,B 0,C 180,E1 -14997.454,E2 -14997.454} C_VEL
LIN {X 0,Y 326.654,Z 279.417,A -85,B 0,C 180,E1 -15000.339,E2 -15000.339} C_VEL
LIN {X 0,Y 326.678,Z 279.418,A -85,B 0,C 180,E1 -15003.141,E2 -15003.141} C_VEL
LIN {X 0,Y 326.644,Z 279.423,A -85,B 0,C 180,E1 -15005.87,E2 -15005.87} C_VEL
LIN {X 0,Y 326.656,Z 279.42,A -85,B 0,C 180,E1 -15009.864,E2 -15009.864} C_VEL
LIN {X 0,Y 326.69,Z 279.412,A -85,B 0,C 180,E1 -15012.471,E2 -15012.471} C_VEL
LIN {X 0,Y 326.751,Z 279.406,A -85,B 0,C 180,E1 -15016.313,E2 -15016.313} C_VEL
LIN {X 0,Y 326.806,Z 279.4,A -85,B 0,C 180,E1 -15020.093,E2 -15020.093} C_VEL
LIN {X 0,Y 326.968,Z 279.375,A -85,B 0,C 180,E1 -15022.589,E2 -15022.589} C_VEL
LIN {X 0,Y 326.977,Z 279.38,A -85,B 0,C 180,E1 -15023.83,E2 -15023.83} C_VEL
LIN {X 0,Y 326.477,Z 279.446,A -85,B 0,C 180,E1 -15027.532,E2 -15027.532} C_VEL
LIN {X 0,Y 326.861,Z 279.869,A -85,B 0,C 180,E1 -15028.767,E2 -15028.767} C_VEL
LIN {X 0,Y 326.114,Z 282.085,A -85,B 0,C 180,E1 -15031.62,E2 -15031.62} C_VEL
LIN {X 0,Y 327.247,Z 285.317,A -85,B 0,C 180,E1 -15031.845,E2 -15031.845} C_VEL
LIN {X 0,Y 333.127,Z 299.082,A -85,B 0,C 180,E1 -15032.946,E2 -15032.946} C_VEL
LIN {X 0,Y 337.802,Z 312.641,A -85,B 0,C 180,E1 -15034.113,E2 -15034.113} C_VEL
LIN {X 0,Y 341.639,Z 326.74,A -85,B 0,C 180,E1 -15035.448,E2 -15035.448} C_VEL
LIN {X 0,Y 341.883,Z 328.211,A -85,B 0,C 180,E1 -15035.592,E2 -15035.592} C_VEL
LIN {X 0,Y 340.083,Z 342.646,A -85,B 0,C 180,E1 -15036.765,E2 -15036.765} C_VEL
LIN {X 0,Y 338.247,Z 355.493,A -85,B 0,C 180,E1 -15038.061,E2 -15038.061} C_VEL
LIN {X 0,Y 336.275,Z 368.148,A -85,B 0,C 180,E1 -15039.624,E2 -15039.624} C_VEL
LIN {X 0,Y 334.464,Z 378.854,A -85,B 0,C 180,E1 -15041.207,E2 -15041.207} C_VEL
LIN {X 0,Y 332.372,Z 389.997,A -85,B 0,C 180,E1 -15043.181,E2 -15043.181} C_VEL
LIN {X 0,Y 330.401,Z 400.331,A -85,B 0,C 180,E1 -15045.419,E2 -15045.419} C_VEL
LIN {X 0,Y 329.01,Z 407.909,A -85,B 0,C 180,E1 -15047.4,E2 -15047.4} C_VEL
LIN {X 0,Y 327.851,Z 414.316,A -85,B 0,C 180,E1 -15049.409,E2 -15049.409} C_VEL
LIN {X 0,Y 326.891,Z 419.735,A -85,B 0,C 180,E1 -15051.437,E2 -15051.437} C_VEL
LIN {X 0,Y 326.194,Z 424.183,A -85,B 0,C 180,E1 -15053.489,E2 -15053.489} C_VEL
LIN {X 0,Y 325.683,Z 427.737,A -85,B 0,C 180,E1 -15055.567,E2 -15055.567} C_VEL
LIN {X 0,Y 325.244,Z 430.444,A -85,B 0,C 180,E1 -15057.636,E2 -15057.636} C_VEL
LIN {X 0,Y 324.984,Z 432.55,A -85,B 0,C 180,E1 -15060.118,E2 -15060.118} C_VEL
LIN {X 0,Y 324.897,Z 433.543,A -85,B 0,C 180,E1 -15062.736,E2 -15062.736} C_VEL
LIN {X 0,Y 324.911,Z 433.499,A -85,B 0,C 180,E1 -15064.722,E2 -15064.722} C_VEL
LIN {X 0,Y 325.145,Z 432.339,A -85,B 0,C 180,E1 -15067.243,E2 -15067.243} C_VEL
LIN {X 0,Y 325.419,Z 430.87,A -85,B 0,C 180,E1 -15068.972,E2 -15068.972} C_VEL
LIN {X 0,Y 325.902,Z 428.391,A -85,B 0,C 180,E1 -15070.998,E2 -15070.998} C_VEL
LIN {X 0,Y 326.688,Z 424.207,A -85,B 0,C 180,E1 -15073.503,E2 -15073.503} C_VEL
LIN {X 0,Y 327.721,Z 418.875,A -85,B 0,C 180,E1 -15075.922,E2 -15075.922} C_VEL
LIN {X 0,Y 329.141,Z 412.037,A -85,B 0,C 180,E1 -15078.359,E2 -15078.359} C_VEL
LIN {X 0,Y 330.855,Z 404.196,A -85,B 0,C 180,E1 -15080.608,E2 -15080.608} C_VEL
LIN {X 0,Y 332.647,Z 395.62,A -85,B 0,C 180,E1 -15082.647,E2 -15082.647} C_VEL
LIN {X 0,Y 334.784,Z 385.693,A -85,B 0,C 180,E1 -15084.599,E2 -15084.599} C_VEL
LIN {X 0,Y 336.797,Z 375.696,A -85,B 0,C 180,E1 -15086.243,E2 -15086.243} C_VEL
LIN {X 0,Y 339.049,Z 363.841,A -85,B 0,C 180,E1 -15087.868,E2 -15087.868} C_VEL
LIN {X 0,Y 340.916,Z 352.485,A -85,B 0,C 180,E1 -15089.169,E2 -15089.169} C_VEL
LIN {X 0,Y 341.283,Z 347.546,A -85,B 0,C 180,E1 -15089.714,E2 -15089.714} C_VEL
LIN {X 0,Y 340.794,Z 342.702,A -85,B 0,C 180,E1 -15090.292,E2 -15090.292} C_VEL
LIN {X 0,Y 338.305,Z 333.256,A -85,B 0,C 180,E1 -15091.478,E2 -15091.478} C_VEL
LIN {X 0,Y 336.332,Z 326.856,A -85,B 0,C 180,E1 -15092.241,E2 -15092.241} C_VEL
LIN {X 0,Y 331.93,Z 313.141,A -85,B 0,C 180,E1 -15093.762,E2 -15093.762} C_VEL
LIN {X 0,Y 326.95,Z 300.772,A -85,B 0,C 180,E1 -15095.095,E2 -15095.095} C_VEL
LIN {X 0,Y 321.168,Z 289.448,A -85,B 0,C 180,E1 -15096.335,E2 -15096.335} C_VEL
LIN {X 0,Y 319.871,Z 286.802,A -85,B 0,C 180,E1 -15096.611,E2 -15096.611} C_VEL
LIN {X 0,Y 319.671,Z 285.875,A -85,B 0,C 180,E1 -15096.69,E2 -15096.69} C_VEL
LIN {X 0,Y 319.889,Z 283.449,A -85,B 0,C 180,E1 -15100.856,E2 -15100.856} C_VEL
LIN {X 0,Y 319.845,Z 281.41,A -85,B 0,C 180,E1 -15104.713,E2 -15104.713} C_VEL
LIN {X 0,Y 319.674,Z 280.291,A -85,B 0,C 180,E1 -15107.301,E2 -15107.301} C_VEL
LIN {X 0,Y 319.875,Z 280.266,A -85,B 0,C 180,E1 -15111.371,E2 -15111.371} C_VEL
LIN {X 0,Y 319.947,Z 280.257,A -85,B 0,C 180,E1 -15113.696,E2 -15113.696} C_VEL
LIN {X 0,Y 319.987,Z 280.25,A -85,B 0,C 180,E1 -15117.484,E2 -15117.484} C_VEL
LIN {X 0,Y 320.146,Z 280.229,A -85,B 0,C 180,E1 -15120.001,E2 -15120.001} C_VEL
LIN {X 0,Y 319.987,Z 280.25,A -85,B 0,C 180,E1 -15122.519,E2 -15122.519} C_VEL
LIN {X 0,Y 319.948,Z 280.253,A -85,B 0,C 180,E1 -15126.307,E2 -15126.307} C_VEL
LIN {X 0,Y 319.839,Z 280.267,A -85,B 0,C 180,E1 -15128.849,E2 -15128.849} C_VEL
LIN {X 0,Y 319.678,Z 280.285,A -85,B 0,C 180,E1 -15132.701,E2 -15132.701} C_VEL
LIN {X 0,Y 319.696,Z 280.283,A -85,B 0,C 180,E1 -15135.297,E2 -15135.297} C_VEL
LIN {X 0,Y 319.672,Z 280.287,A -85,B 0,C 180,E1 -15139.256,E2 -15139.256} C_VEL
LIN {X 0,Y 319.568,Z 280.301,A -85,B 0,C 180,E1 -15143.321,E2 -15143.321} C_VEL
LIN {X 0,Y 319.633,Z 280.296,A -85,B 0,C 180,E1 -15146.089,E2 -15146.089} C_VEL
LIN {X 0,Y 319.616,Z 280.371,A -85,B 0,C 180,E1 -15147.502,E2 -15147.502} C_VEL
LIN {X 0,Y 320.016,Z 282.854,A -85,B 0,C 180,E1 -15151.077,E2 -15151.077} C_VEL
LIN {X 0,Y 320.548,Z 285.901,A -85,B 0,C 180,E1 -15154.755,E2 -15154.755} C_VEL
LIN {X 0,Y 321.108,Z 288.992,A -85,B 0,C 180,E1 -15158.01,E2 -15158.01} C_VEL
LIN {X 0,Y 321.817,Z 293.333,A -85,B 0,C 180,E1 -15162.056,E2 -15162.056} C_VEL
LIN {X 0,Y 322.656,Z 298.046,A -85,B 0,C 180,E1 -15165.956,E2 -15165.956} C_VEL
LIN {X 0,Y 322.713,Z 301.457,A -85,B 0,C 180,E1 -15168.485,E2 -15168.485} C_VEL
LIN {X 0,Y 321.764,Z 307.129,A -85,B 0,C 180,E1 -15172.298,E2 -15172.298} C_VEL
LIN {X 0,Y 321.098,Z 311.865,A -85,B 0,C 180,E1 -15175.316,E2 -15175.316} C_VEL
LIN {X 0,Y 320.869,Z 313.678,A -85,B 0,C 180,E1 -15176.447,E2 -15176.447} C_VEL
LIN {X 0,Y 321.753,Z 316.917,A -85,B 0,C 180,E1 -15176.67,E2 -15176.67} C_VEL
LIN {X 0,Y 326.411,Z 330.188,A -85,B 0,C 180,E1 -15177.773,E2 -15177.773} C_VEL
LIN {X 0,Y 330.296,Z 345.092,A -85,B 0,C 180,E1 -15179.035,E2 -15179.035} C_VEL
LIN {X 0,Y 332.83,Z 360.016,A -85,B 0,C 180,E1 -15180.372,E2 -15180.372} C_VEL
LIN {X 0,Y 334.283,Z 375.034,A -85,B 0,C 180,E1 -15181.855,E2 -15181.855} C_VEL
LIN {X 0,Y 334.286,Z 378.462,A -85,B 0,C 180,E1 -15182.197,E2 -15182.197} C_VEL
LIN {X 0,Y 331.856,Z 392.463,A -85,B 0,C 180,E1 -15183.595,E2 -15183.595} C_VEL
LIN {X 0,Y 329.466,Z 404.704,A -85,B 0,C 180,E1 -15185.085,E2 -15185.085} C_VEL
LIN {X 0,Y 326.941,Z 416.994,A -85,B 0,C 180,E1 -15186.903,E2 -15186.903} C_VEL
LIN {X 0,Y 324.835,Z 427.351,A -85,B 0,C 180,E1 -15188.754,E2 -15188.754} C_VEL
LIN {X 0,Y 322.767,Z 437.554,A -85,B 0,C 180,E1 -15190.938,E2 -15190.938} C_VEL
LIN {X 0,Y 321.142,Z 446.075,A -85,B 0,C 180,E1 -15193.145,E2 -15193.145} C_VEL
LIN {X 0,Y 319.696,Z 453.499,A -85,B 0,C 180,E1 -15195.468,E2 -15195.468} C_VEL
LIN {X 0,Y 318.882,Z 459.833,A -85,B 0,C 180,E1 -15197.915,E2 -15197.915} C_VEL
LIN {X 0,Y 318.225,Z 465.045,A -85,B 0,C 180,E1 -15200.467,E2 -15200.467} C_VEL
LIN {X 0,Y 318.023,Z 468.1,A -85,B 0,C 180,E1 -15202.381,E2 -15202.381} C_VEL
LIN {X 0,Y 317.998,Z 470.161,A -85,B 0,C 180,E1 -15204.012,E2 -15204.012} C_VEL
LIN {X 0,Y 317.899,Z 472.074,A -85,B 0,C 180,E1 -15206.198,E2 -15206.198} C_VEL
LIN {X 0,Y 317.936,Z 473.239,A -85,B 0,C 180,E1 -15208.734,E2 -15208.734} C_VEL
LIN {X 0,Y 317.994,Z 473.387,A -85,B 0,C 180,E1 -15210.001,E2 -15210.001} C_VEL
LIN {X 0,Y 317.871,Z 472.765,A -85,B 0,C 180,E1 -15212.535,E2 -15212.535} C_VEL
LIN {X 0,Y 317.918,Z 470.922,A -85,B 0,C 180,E1 -15215.074,E2 -15215.074} C_VEL
LIN {X 0,Y 318.014,Z 467.862,A -85,B 0,C 180,E1 -15217.621,E2 -15217.621} C_VEL
LIN {X 0,Y 318.356,Z 463.525,A -85,B 0,C 180,E1 -15220.173,E2 -15220.173} C_VEL
LIN {X 0,Y 319.057,Z 457.802,A -85,B 0,C 180,E1 -15222.726,E2 -15222.726} C_VEL
LIN {X 0,Y 320.132,Z 450.541,A -85,B 0,C 180,E1 -15225.275,E2 -15225.275} C_VEL
LIN {X 0,Y 321.501,Z 442.784,A -85,B 0,C 180,E1 -15227.493,E2 -15227.493} C_VEL
LIN {X 0,Y 323.314,Z 433.466,A -85,B 0,C 180,E1 -15229.691,E2 -15229.691} C_VEL
LIN {X 0,Y 325.1,Z 423.629,A -85,B 0,C 180,E1 -15231.63,E2 -15231.63} C_VEL
LIN {X 0,Y 327.409,Z 411.702,A -85,B 0,C 180,E1 -15233.566,E2 -15233.566} C_VEL
LIN {X 0,Y 329.649,Z 399.198,A -85,B 0,C 180,E1 -15235.24,E2 -15235.24} C_VEL
LIN {X 0,Y 332.027,Z 385.858,A -85,B 0,C 180,E1 -15236.685,E2 -15236.685} C_VEL
LIN {X 0,Y 333.344,Z 377.45,A -85,B 0,C 180,E1 -15237.45,E2 -15237.45} C_VEL
LIN {X 0,Y 332.887,Z 371.175,A -85,B 0,C 180,E1 -15238.068,E2 -15238.068} C_VEL
LIN {X 0,Y 330.756,Z 356.543,A -85,B 0,C 180,E1 -15239.403,E2 -15239.403} C_VEL
LIN {X 0,Y 327.527,Z 340.76,A -85,B 0,C 180,E1 -15240.654,E2 -15240.654} C_VEL
LIN {X 0,Y 323.37,Z 325.222,A -85,B 0,C 180,E1 -15241.726,E2 -15241.726} C_VEL
LIN {X 0,Y 320.725,Z 316.797,A -85,B 0,C 180,E1 -15242.247,E2 -15242.247} C_VEL
LIN {X 0,Y 320.644,Z 316.044,A -85,B 0,C 180,E1 -15242.308,E2 -15242.308} C_VEL
LIN {X 0,Y 321.453,Z 309.657,A -85,B 0,C 180,E1 -15246.18,E2 -15246.18} C_VEL
LIN {X 0,Y 322.186,Z 304.737,A -85,B 0,C 180,E1 -15249.243,E2 -15249.243} C_VEL
LIN {X 0,Y 322.668,Z 301.254,A -85,B 0,C 180,E1 -15251.507,E2 -15251.507} C_VEL
LIN {X 0,Y 322.605,Z 297.316,A -85,B 0,C 180,E1 -15254.198,E2 -15254.198} C_VEL
LIN {X 0,Y 321.668,Z 292.25,A -85,B 0,C 180,E1 -15257.976,E2 -15257.976} C_VEL
LIN {X 0,Y 320.735,Z 287,A -85,B 0,C 180,E1 -15262.153,E2 -15262.153} C_VEL
LIN {X 0,Y 320.133,Z 283.452,A -85,B 0,C 180,E1 -15265.194,E2 -15265.194} C_VEL
LIN {X 0,Y 319.567,Z 280.305,A -85,B 0,C 180,E1 -15268.141,E2 -15268.141} C_VEL
LIN {X 0,Y 319.617,Z 280.298,A -85,B 0,C 180,E1 -15271.59,E2 -15271.59} C_VEL
LIN {X 0,Y 319.611,Z 280.298,A -85,B 0,C 180,E1 -15275.303,E2 -15275.303} C_VEL
LIN {X 0,Y 319.604,Z 280.298,A -85,B 0,C 180,E1 -15278.047,E2 -15278.047} C_VEL
LIN {X 0,Y 319.695,Z 280.288,A -85,B 0,C 180,E1 -15280.961,E2 -15280.961} C_VEL
LIN {X 0,Y 319.737,Z 280.281,A -85,B 0,C 180,E1 -15285.275,E2 -15285.275} C_VEL
LIN {X 0,Y 319.757,Z 280.278,A -85,B 0,C 180,E1 -15289.872,E2 -15289.872} C_VEL
LIN {X 0,Y 319.914,Z 280.258,A -85,B 0,C 180,E1 -15293.693,E2 -15293.693} C_VEL
LIN {X 0,Y 319.994,Z 280.248,A -85,B 0,C 180,E1 -15297.481,E2 -15297.481} C_VEL
LIN {X 0,Y 320.155,Z 280.229,A -85,B 0,C 180,E1 -15299.999,E2 -15299.999} C_VEL
LIN {X 0,Y 319.993,Z 280.249,A -85,B 0,C 180,E1 -15302.516,E2 -15302.516} C_VEL
LIN {X 0,Y 319.934,Z 280.254,A -85,B 0,C 180,E1 -15306.666,E2 -15306.666} C_VEL
LIN {X 0,Y 319.761,Z 280.28,A -85,B 0,C 180,E1 -15310.126,E2 -15310.126} C_VEL
LIN {X 0,Y 319.733,Z 280.281,A -85,B 0,C 180,E1 -15314.722,E2 -15314.722} C_VEL
LIN {X 0,Y 319.691,Z 280.282,A -85,B 0,C 180,E1 -15319.036,E2 -15319.036} C_VEL
LIN {X 0,Y 319.571,Z 280.3,A -85,B 0,C 180,E1 -15323.318,E2 -15323.318} C_VEL
LIN {X 0,Y 319.634,Z 280.295,A -85,B 0,C 180,E1 -15326.086,E2 -15326.086} C_VEL
LIN {X 0,Y 319.579,Z 280.296,A -85,B 0,C 180,E1 -15328.933,E2 -15328.933} C_VEL
LIN {X 0,Y 319.53,Z 280.309,A -85,B 0,C 180,E1 -15331.86,E2 -15331.86} C_VEL
LIN {X 0,Y 319.578,Z 280.298,A -85,B 0,C 180,E1 -15335.541,E2 -15335.541} C_VEL
LIN {X 0,Y 319.57,Z 280.305,A -85,B 0,C 180,E1 -15338.006,E2 -15338.006} C_VEL
LIN {X 0,Y 319.551,Z 280.305,A -85,B 0,C 180,E1 -15341.601,E2 -15341.601} C_VEL
LIN {X 0,Y 319.579,Z 280.299,A -85,B 0,C 180,E1 -15345.272,E2 -15345.272} C_VEL
LIN {X 0,Y 319.575,Z 280.297,A -85,B 0,C 180,E1 -15348.718,E2 -15348.718} C_VEL
LIN {X 0,Y 319.593,Z 280.298,A -85,B 0,C 180,E1 -15352.338,E2 -15352.338} C_VEL
LIN {X 0,Y 319.554,Z 280.301,A -85,B 0,C 180,E1 -15355.122,E2 -15355.122} C_VEL
LIN {X 0,Y 319.563,Z 280.302,A -85,B 0,C 180,E1 -15359.056,E2 -15359.056} C_VEL
LIN {X 0,Y 319.61,Z 280.297,A -85,B 0,C 180,E1 -15362.497,E2 -15362.497} C_VEL
LIN {X 0,Y 319.597,Z 280.299,A -85,B 0,C 180,E1 -15365.303,E2 -15365.303} C_VEL
LIN {X 0,Y 319.589,Z 280.299,A -85,B 0,C 180,E1 -15368.046,E2 -15368.046} C_VEL
LIN {X 0,Y 319.681,Z 280.288,A -85,B 0,C 180,E1 -15370.961,E2 -15370.961} C_VEL
LIN {X 0,Y 319.722,Z 280.286,A -85,B 0,C 180,E1 -15375.275,E2 -15375.275} C_VEL
LIN {X 0,Y 319.75,Z 280.28,A -85,B 0,C 180,E1 -15379.872,E2 -15379.872} C_VEL
LIN {X 0,Y 319.922,Z 280.251,A -85,B 0,C 180,E1 -15382.425,E2 -15382.425} C_VEL
LIN {X 0,Y 319.934,Z 280.258,A -85,B 0,C 180,E1 -15383.693,E2 -15383.693} C_VEL
LIN {X 0,Y 319.426,Z 280.324,A -85,B 0,C 180,E1 -15387.477,E2 -15387.477} C_VEL
LIN {X 0,Y 319.822,Z 280.824,A -85,B 0,C 180,E1 -15388.74,E2 -15388.74} C_VEL
LIN {X 0,Y 319.214,Z 282.696,A -85,B 0,C 180,E1 -15390.945,E2 -15390.945} C_VEL
LIN {X 0,Y 320.356,Z 285.838,A -85,B 0,C 180,E1 -15391.166,E2 -15391.166} C_VEL
LIN {X 0,Y 326.282,Z 299.677,A -85,B 0,C 180,E1 -15392.314,E2 -15392.314} C_VEL
LIN {X 0,Y 330.922,Z 313.005,A -85,B 0,C 180,E1 -15393.5,E2 -15393.5} C_VEL
LIN {X 0,Y 334.65,Z 326.492,A -85,B 0,C 180,E1 -15394.818,E2 -15394.818} C_VEL
LIN {X 0,Y 335.326,Z 330.039,A -85,B 0,C 180,E1 -15395.179,E2 -15395.179} C_VEL
LIN {X 0,Y 333.511,Z 344.1,A -85,B 0,C 180,E1 -15396.366,E2 -15396.366} C_VEL
LIN {X 0,Y 331.498,Z 357.454,A -85,B 0,C 180,E1 -15397.767,E2 -15397.767} C_VEL
LIN {X 0,Y 329.441,Z 369.872,A -85,B 0,C 180,E1 -15399.361,E2 -15399.361} C_VEL
LIN {X 0,Y 327.376,Z 381.344,A -85,B 0,C 180,E1 -15401.139,E2 -15401.139} C_VEL
LIN {X 0,Y 325.524,Z 390.985,A -85,B 0,C 180,E1 -15402.916,E2 -15402.916} C_VEL
LIN {X 0,Y 323.544,Z 400.874,A -85,B 0,C 180,E1 -15405.108,E2 -15405.108} C_VEL
LIN {X 0,Y 322.093,Z 408.447,A -85,B 0,C 180,E1 -15407.13,E2 -15407.13} C_VEL
LIN {X 0,Y 320.689,Z 415.916,A -85,B 0,C 180,E1 -15409.555,E2 -15409.555} C_VEL
LIN {X 0,Y 319.642,Z 421.814,A -85,B 0,C 180,E1 -15411.948,E2 -15411.948} C_VEL
LIN {X 0,Y 318.951,Z 425.955,A -85,B 0,C 180,E1 -15414.056,E2 -15414.056} C_VEL
LIN {X 0,Y 318.453,Z 429.251,A -85,B 0,C 180,E1 -15416.191,E2 -15416.191} C_VEL
LIN {X 0,Y 317.967,Z 432.326,A -85,B 0,C 180,E1 -15419.094,E2 -15419.094} C_VEL
LIN {X 0,Y 317.874,Z 433.289,A -85,B 0,C 180,E1 -15420.564,E2 -15420.564} C_VEL
LIN {X 0,Y 317.808,Z 433.998,A -85,B 0,C 180,E1 -15422.828,E2 -15422.828} C_VEL
LIN {X 0,Y 317.857,Z 433.843,A -85,B 0,C 180,E1 -15425.109,E2 -15425.109} C_VEL
LIN {X 0,Y 318.085,Z 432.827,A -85,B 0,C 180,E1 -15427.309,E2 -15427.309} C_VEL
LIN {X 0,Y 318.509,Z 430.626,A -85,B 0,C 180,E1 -15429.783,E2 -15429.783} C_VEL
LIN {X 0,Y 319.167,Z 427.404,A -85,B 0,C 180,E1 -15432.191,E2 -15432.191} C_VEL
LIN {X 0,Y 320.041,Z 422.961,A -85,B 0,C 180,E1 -15434.643,E2 -15434.643} C_VEL
LIN {X 0,Y 321.153,Z 417.93,A -85,B 0,C 180,E1 -15436.809,E2 -15436.809} C_VEL
LIN {X 0,Y 322.696,Z 411.013,A -85,B 0,C 180,E1 -15439.206,E2 -15439.206} C_VEL
LIN {X 0,Y 324.368,Z 403.764,A -85,B 0,C 180,E1 -15441.259,E2 -15441.259} C_VEL
LIN {X 0,Y 326.288,Z 394.934,A -85,B 0,C 180,E1 -15443.352,E2 -15443.352} C_VEL
LIN {X 0,Y 328.621,Z 384.317,A -85,B 0,C 180,E1 -15445.421,E2 -15445.421} C_VEL
LIN {X 0,Y 331.058,Z 372.79,A -85,B 0,C 180,E1 -15447.264,E2 -15447.264} C_VEL
LIN {X 0,Y 333.449,Z 360.188,A -85,B 0,C 180,E1 -15448.927,E2 -15448.927} C_VEL
LIN {X 0,Y 335.717,Z 346.718,A -85,B 0,C 180,E1 -15450.374,E2 -15450.374} C_VEL
LIN {X 0,Y 337.764,Z 332.68,A -85,B 0,C 180,E1 -15451.579,E2 -15451.579} C_VEL
LIN {X 0,Y 336.332,Z 326.856,A -85,B 0,C 180,E1 -15452.241,E2 -15452.241} C_VEL
LIN {X 0,Y 334.425,Z 322.407,A -85,B 0,C 180,E1 -15452.817,E2 -15452.817} C_VEL
LIN {X 0,Y 329.641,Z 316.107,A -85,B 0,C 180,E1 -15453.847,E2 -15453.847} C_VEL
LIN {X 0,Y 325.487,Z 311.213,A -85,B 0,C 180,E1 -15454.685,E2 -15454.685} C_VEL
LIN {X 0,Y 322.774,Z 307.103,A -85,B 0,C 180,E1 -15455.283,E2 -15455.283} C_VEL
LIN {X 0,Y 322.015,Z 305.587,A -85,B 0,C 180,E1 -15455.468,E2 -15455.468} C_VEL
LIN {X 0,Y 316.399,Z 294,A -85,B 0,C 180,E1 -15456.827,E2 -15456.827} C_VEL
LIN {X 0,Y 314.307,Z 290.102,A -85,B 0,C 180,E1 -15457.273,E2 -15457.273} C_VEL
LIN {X 0,Y 312.887,Z 287.112,A -85,B 0,C 180,E1 -15457.597,E2 -15457.597} C_VEL
LIN {X 0,Y 312.76,Z 286.447,A -85,B 0,C 180,E1 -15457.674,E2 -15457.674} C_VEL
LIN {X 0,Y 312.879,Z 284.232,A -85,B 0,C 180,E1 -15461.673,E2 -15461.673} C_VEL
LIN {X 0,Y 312.822,Z 282.221,A -85,B 0,C 180,E1 -15465.694,E2 -15465.694} C_VEL
LIN {X 0,Y 312.662,Z 281.164,A -85,B 0,C 180,E1 -15468.33,E2 -15468.33} C_VEL
LIN {X 0,Y 312.866,Z 281.138,A -85,B 0,C 180,E1 -15472.256,E2 -15472.256} C_VEL
LIN {X 0,Y 312.714,Z 281.158,A -85,B 0,C 180,E1 -15474.844,E2 -15474.844} C_VEL
LIN {X 0,Y 312.986,Z 281.125,A -85,B 0,C 180,E1 -15478.715,E2 -15478.715} C_VEL
LIN {X 0,Y 312.986,Z 281.123,A -85,B 0,C 180,E1 -15481.288,E2 -15481.288} C_VEL
LIN {X 0,Y 312.715,Z 281.159,A -85,B 0,C 180,E1 -15485.159,E2 -15485.159} C_VEL
LIN {X 0,Y 312.868,Z 281.138,A -85,B 0,C 180,E1 -15487.747,E2 -15487.747} C_VEL
LIN {X 0,Y 312.666,Z 281.163,A -85,B 0,C 180,E1 -15491.673,E2 -15491.673} C_VEL
LIN {X 0,Y 312.697,Z 281.155,A -85,B 0,C 180,E1 -15494.889,E2 -15494.889} C_VEL
LIN {X 0,Y 312.628,Z 281.164,A -85,B 0,C 180,E1 -15499.238,E2 -15499.238} C_VEL
LIN {X 0,Y 312.543,Z 281.178,A -85,B 0,C 180,E1 -15502.791,E2 -15502.791} C_VEL
LIN {X 0,Y 312.601,Z 281.171,A -85,B 0,C 180,E1 -15505.937,E2 -15505.937} C_VEL
LIN {X 0,Y 312.927,Z 283.425,A -85,B 0,C 180,E1 -15509.611,E2 -15509.611} C_VEL
LIN {X 0,Y 313.289,Z 285.652,A -85,B 0,C 180,E1 -15512.575,E2 -15512.575} C_VEL
LIN {X 0,Y 313.872,Z 288.841,A -85,B 0,C 180,E1 -15516.287,E2 -15516.287} C_VEL
LIN {X 0,Y 314.53,Z 292.921,A -85,B 0,C 180,E1 -15520.391,E2 -15520.391} C_VEL
LIN {X 0,Y 315.195,Z 296.66,A -85,B 0,C 180,E1 -15523.728,E2 -15523.728} C_VEL
LIN {X 0,Y 315.75,Z 299.863,A -85,B 0,C 180,E1 -15526.371,E2 -15526.371} C_VEL
LIN {X 0,Y 315.743,Z 302.175,A -85,B 0,C 180,E1 -15528.107,E2 -15528.107} C_VEL
LIN {X 0,Y 314.959,Z 306.822,A -85,B 0,C 180,E1 -15531.353,E2 -15531.353} C_VEL
LIN {X 0,Y 314.079,Z 312.672,A -85,B 0,C 180,E1 -15535.208,E2 -15535.208} C_VEL
LIN {X 0,Y 314.035,Z 313.304,A -85,B 0,C 180,E1 -15535.503,E2 -15535.503} C_VEL
LIN {X 0,Y 315.082,Z 316.716,A -85,B 0,C 180,E1 -15535.762,E2 -15535.762} C_VEL
LIN {X 0,Y 319.08,Z 327.793,A -85,B 0,C 180,E1 -15536.744,E2 -15536.744} C_VEL
LIN {X 0,Y 322.819,Z 340.859,A -85,B 0,C 180,E1 -15537.905,E2 -15537.905} C_VEL
LIN {X 0,Y 325.477,Z 353.943,A -85,B 0,C 180,E1 -15539.105,E2 -15539.105} C_VEL
LIN {X 0,Y 327.075,Z 367.038,A -85,B 0,C 180,E1 -15540.383,E2 -15540.383} C_VEL
LIN {X 0,Y 327.894,Z 379.12,A -85,B 0,C 180,E1 -15541.675,E2 -15541.675} C_VEL
LIN {X 0,Y 325.495,Z 392.409,A -85,B 0,C 180,E1 -15543.037,E2 -15543.037} C_VEL
LIN {X 0,Y 322.978,Z 404.588,A -85,B 0,C 180,E1 -15544.549,E2 -15544.549} C_VEL
LIN {X 0,Y 320.356,Z 416.816,A -85,B 0,C 180,E1 -15546.4,E2 -15546.4} C_VEL
LIN {X 0,Y 318.008,Z 427.771,A -85,B 0,C 180,E1 -15548.412,E2 -15548.412} C_VEL
LIN {X 0,Y 316.006,Z 437.268,A -85,B 0,C 180,E1 -15550.513,E2 -15550.513} C_VEL
LIN {X 0,Y 314.254,Z 445.751,A -85,B 0,C 180,E1 -15552.764,E2 -15552.764} C_VEL
LIN {X 0,Y 312.812,Z 452.868,A -85,B 0,C 180,E1 -15555.038,E2 -15555.038} C_VEL
LIN {X 0,Y 311.852,Z 459.464,A -85,B 0,C 180,E1 -15557.639,E2 -15557.639} C_VEL
LIN {X 0,Y 311.181,Z 464.66,A -85,B 0,C 180,E1 -15560.249,E2 -15560.249} C_VEL
LIN {X 0,Y 310.958,Z 467.705,A -85,B 0,C 180,E1 -15562.207,E2 -15562.207} C_VEL
LIN {X 0,Y 310.824,Z 470.637,A -85,B 0,C 180,E1 -15564.812,E2 -15564.812} C_VEL
LIN {X 0,Y 310.792,Z 472.371,A -85,B 0,C 180,E1 -15567.409,E2 -15567.409} C_VEL
LIN {X 0,Y 310.907,Z 472.944,A -85,B 0,C 180,E1 -15570.001,E2 -15570.001} C_VEL
LIN {X 0,Y 310.788,Z 472.316,A -85,B 0,C 180,E1 -15572.593,E2 -15572.593} C_VEL
LIN {X 0,Y 310.837,Z 470.457,A -85,B 0,C 180,E1 -15575.19,E2 -15575.19} C_VEL
LIN {X 0,Y 310.956,Z 467.381,A -85,B 0,C 180,E1 -15577.795,E2 -15577.795} C_VEL
LIN {X 0,Y 311.305,Z 463.02,A -85,B 0,C 180,E1 -15580.406,E2 -15580.406} C_VEL
LIN {X 0,Y 312.039,Z 457.27,A -85,B 0,C 180,E1 -15583.017,E2 -15583.017} C_VEL
LIN {X 0,Y 313.201,Z 449.979,A -85,B 0,C 180,E1 -15585.622,E2 -15585.622} C_VEL
LIN {X 0,Y 314.647,Z 442.184,A -85,B 0,C 180,E1 -15587.887,E2 -15587.887} C_VEL
LIN {X 0,Y 316.559,Z 432.823,A -85,B 0,C 180,E1 -15590.129,E2 -15590.129} C_VEL
LIN {X 0,Y 318.364,Z 423.301,A -85,B 0,C 180,E1 -15592.043,E2 -15592.043} C_VEL
LIN {X 0,Y 320.63,Z 412.021,A -85,B 0,C 180,E1 -15593.924,E2 -15593.924} C_VEL
LIN {X 0,Y 322.946,Z 399.666,A -85,B 0,C 180,E1 -15595.629,E2 -15595.629} C_VEL
LIN {X 0,Y 325.391,Z 386.5,A -85,B 0,C 180,E1 -15597.102,E2 -15597.102} C_VEL
LIN {X 0,Y 326.758,Z 377.318,A -85,B 0,C 180,E1 -15597.97,E2 -15597.97} C_VEL
LIN {X 0,Y 325.125,Z 363.479,A -85,B 0,C 180,E1 -15599.357,E2 -15599.357} C_VEL
LIN {X 0,Y 322.765,Z 349.64,A -85,B 0,C 180,E1 -15600.581,E2 -15600.581} C_VEL
LIN {X 0,Y 319.016,Z 333.714,A -85,B 0,C 180,E1 -15601.811,E2 -15601.811} C_VEL
LIN {X 0,Y 314.592,Z 318.968,A -85,B 0,C 180,E1 -15602.813,E2 -15602.813} C_VEL
LIN {X 0,Y 313.732,Z 315.595,A -85,B 0,C 180,E1 -15603.055,E2 -15603.055} C_VEL
LIN {X 0,Y 314.644,Z 309.124,A -85,B 0,C 180,E1 -15607.092,E2 -15607.092} C_VEL
LIN {X 0,Y 315.486,Z 303.451,A -85,B 0,C 180,E1 -15610.763,E2 -15610.763} C_VEL
LIN {X 0,Y 315.673,Z 299.27,A -85,B 0,C 180,E1 -15613.645,E2 -15613.645} C_VEL
LIN {X 0,Y 315.071,Z 295.759,A -85,B 0,C 180,E1 -15616.251,E2 -15616.251} C_VEL
LIN {X 0,Y 314.304,Z 291.526,A -85,B 0,C 180,E1 -15619.574,E2 -15619.574} C_VEL
LIN {X 0,Y 313.454,Z 286.43,A -85,B 0,C 180,E1 -15623.821,E2 -15623.821} C_VEL
LIN {X 0,Y 312.767,Z 282.535,A -85,B 0,C 180,E1 -15627.364,E2 -15627.364} C_VEL
LIN {X 0,Y 312.534,Z 281.181,A -85,B 0,C 180,E1 -15628.854,E2 -15628.854} C_VEL
LIN {X 0,Y 312.576,Z 281.175,A -85,B 0,C 180,E1 -15631.824,E2 -15631.824} C_VEL
LIN {X 0,Y 312.592,Z 281.176,A -85,B 0,C 180,E1 -15634.71,E2 -15634.71} C_VEL
LIN {X 0,Y 312.594,Z 281.171,A -85,B 0,C 180,E1 -15637.528,E2 -15637.528} C_VEL
LIN {X 0,Y 312.645,Z 281.164,A -85,B 0,C 180,E1 -15641.656,E2 -15641.656} C_VEL
LIN {X 0,Y 312.7,Z 281.157,A -85,B 0,C 180,E1 -15645.685,E2 -15645.685} C_VEL
LIN {X 0,Y 312.703,Z 281.157,A -85,B 0,C 180,E1 -15649.641,E2 -15649.641} C_VEL
LIN {X 0,Y 312.822,Z 281.145,A -85,B 0,C 180,E1 -15652.252,E2 -15652.252} C_VEL
LIN {X 0,Y 312.711,Z 281.158,A -85,B 0,C 180,E1 -15654.841,E2 -15654.841} C_VEL
LIN {X 0,Y 312.995,Z 281.122,A -85,B 0,C 180,E1 -15658.712,E2 -15658.712} C_VEL
LIN {X 0,Y 312.995,Z 281.119,A -85,B 0,C 180,E1 -15661.285,E2 -15661.285} C_VEL
LIN {X 0,Y 312.72,Z 281.15,A -85,B 0,C 180,E1 -15665.156,E2 -15665.156} C_VEL
LIN {X 0,Y 312.875,Z 281.135,A -85,B 0,C 180,E1 -15667.744,E2 -15667.744} C_VEL
LIN {X 0,Y 312.672,Z 281.156,A -85,B 0,C 180,E1 -15671.67,E2 -15671.67} C_VEL
LIN {X 0,Y 312.702,Z 281.156,A -85,B 0,C 180,E1 -15674.886,E2 -15674.886} C_VEL
LIN {X 0,Y 312.632,Z 281.161,A -85,B 0,C 180,E1 -15679.235,E2 -15679.235} C_VEL
LIN {X 0,Y 312.546,Z 281.175,A -85,B 0,C 180,E1 -15682.787,E2 -15682.787} C_VEL
LIN {X 0,Y 312.602,Z 281.172,A -85,B 0,C 180,E1 -15685.934,E2 -15685.934} C_VEL
LIN {X 0,Y 312.537,Z 281.175,A -85,B 0,C 180,E1 -15689.649,E2 -15689.649} C_VEL
LIN {X 0,Y 312.518,Z 281.181,A -85,B 0,C 180,E1 -15693.687,E2 -15693.687} C_VEL
LIN {X 0,Y 312.535,Z 281.175,A -85,B 0,C 180,E1 -15697.382,E2 -15697.382} C_VEL
LIN {X 0,Y 312.488,Z 281.182,A -85,B 0,C 180,E1 -15700.707,E2 -15700.707} C_VEL
LIN {X 0,Y 312.521,Z 281.18,A -85,B 0,C 180,E1 -15704.195,E2 -15704.195} C_VEL
LIN {X 0,Y 312.545,Z 281.177,A -85,B 0,C 180,E1 -15707.903,E2 -15707.903} C_VEL
LIN {X 0,Y 312.552,Z 281.179,A -85,B 0,C 180,E1 -15711.903,E2 -15711.903} C_VEL
LIN {X 0,Y 312.5,Z 281.184,A -85,B 0,C 180,E1 -15715.788,E2 -15715.788} C_VEL
LIN {X 0,Y 312.517,Z 281.18,A -85,B 0,C 180,E1 -15718.852,E2 -15718.852} C_VEL
LIN {X 0,Y 312.578,Z 281.176,A -85,B 0,C 180,E1 -15721.824,E2 -15721.824} C_VEL
LIN {X 0,Y 312.578,Z 281.17,A -85,B 0,C 180,E1 -15724.709,E2 -15724.709} C_VEL
LIN {X 0,Y 312.579,Z 281.177,A -85,B 0,C 180,E1 -15727.527,E2 -15727.527} C_VEL
LIN {X 0,Y 312.63,Z 281.167,A -85,B 0,C 180,E1 -15731.655,E2 -15731.655} C_VEL
LIN {X 0,Y 312.685,Z 281.161,A -85,B 0,C 180,E1 -15735.685,E2 -15735.685} C_VEL
LIN {X 0,Y 312.694,Z 281.161,A -85,B 0,C 180,E1 -15739.641,E2 -15739.641} C_VEL
LIN {X 0,Y 312.861,Z 281.13,A -85,B 0,C 180,E1 -15742.253,E2 -15742.253} C_VEL
LIN {X 0,Y 312.894,Z 281.134,A -85,B 0,C 180,E1 -15743.551,E2 -15743.551} C_VEL
LIN {X 0,Y 312.377,Z 281.203,A -85,B 0,C 180,E1 -15747.42,E2 -15747.42} C_VEL
LIN {X 0,Y 312.783,Z 281.803,A -85,B 0,C 180,E1 -15748.712,E2 -15748.712} C_VEL
LIN {X 0,Y 312.4,Z 282.921,A -85,B 0,C 180,E1 -15750.201,E2 -15750.201} C_VEL
LIN {X 0,Y 314.444,Z 288.8,A -85,B 0,C 180,E1 -15750.64,E2 -15750.64} C_VEL
LIN {X 0,Y 320.914,Z 304.197,A -85,B 0,C 180,E1 -15752.009,E2 -15752.009} C_VEL
LIN {X 0,Y 325.591,Z 318.431,A -85,B 0,C 180,E1 -15753.366,E2 -15753.366} C_VEL
LIN {X 0,Y 328.661,Z 330.341,A -85,B 0,C 180,E1 -15754.604,E2 -15754.604} C_VEL
LIN {X 0,Y 328.336,Z 335.752,A -85,B 0,C 180,E1 -15755.065,E2 -15755.065} C_VEL
LIN {X 0,Y 326.356,Z 349.541,A -85,B 0,C 180,E1 -15756.349,E2 -15756.349} C_VEL
LIN {X 0,Y 324.316,Z 362.074,A -85,B 0,C 180,E1 -15757.783,E2 -15757.783} C_VEL
LIN {X 0,Y 322.254,Z 373.819,A -85,B 0,C 180,E1 -15759.413,E2 -15759.413} C_VEL
LIN {X 0,Y 319.939,Z 385.679,A -85,B 0,C 180,E1 -15761.402,E2 -15761.402} C_VEL
LIN {X 0,Y 317.917,Z 395.694,A -85,B 0,C 180,E1 -15763.432,E2 -15763.432} C_VEL
LIN {X 0,Y 315.907,Z 405.148,A -85,B 0,C 180,E1 -15765.753,E2 -15765.753} C_VEL
LIN {X 0,Y 314.344,Z 413.355,A -85,B 0,C 180,E1 -15768.24,E2 -15768.24} C_VEL
LIN {X 0,Y 313.184,Z 419.053,A -85,B 0,C 180,E1 -15770.353,E2 -15770.353} C_VEL
LIN {X 0,Y 312.283,Z 424.159,A -85,B 0,C 180,E1 -15772.679,E2 -15772.679} C_VEL
LIN {X 0,Y 311.522,Z 428.915,A -85,B 0,C 180,E1 -15775.528,E2 -15775.528} C_VEL
LIN {X 0,Y 310.972,Z 432.13,A -85,B 0,C 180,E1 -15778.332,E2 -15778.332} C_VEL
LIN {X 0,Y 310.777,Z 433.817,A -85,B 0,C 180,E1 -15780.761,E2 -15780.761} C_VEL
LIN {X 0,Y 310.752,Z 434.497,A -85,B 0,C 180,E1 -15783.2,E2 -15783.2} C_VEL
LIN {X 0,Y 310.826,Z 434.031,A -85,B 0,C 180,E1 -15786.005,E2 -15786.005} C_VEL
LIN {X 0,Y 311.053,Z 433.099,A -85,B 0,C 180,E1 -15787.743,E2 -15787.743} C_VEL
LIN {X 0,Y 311.475,Z 431.155,A -85,B 0,C 180,E1 -15789.903,E2 -15789.903} C_VEL
LIN {X 0,Y 312.184,Z 427.794,A -85,B 0,C 180,E1 -15792.482,E2 -15792.482} C_VEL
LIN {X 0,Y 313.127,Z 423.332,A -85,B 0,C 180,E1 -15794.99,E2 -15794.99} C_VEL
LIN {X 0,Y 314.49,Z 417.501,A -85,B 0,C 180,E1 -15797.514,E2 -15797.514} C_VEL
LIN {X 0,Y 316.114,Z 410.721,A -85,B 0,C 180,E1 -15799.856,E2 -15799.856} C_VEL
LIN {X 0,Y 318.246,Z 401.756,A -85,B 0,C 180,E1 -15802.353,E2 -15802.353} C_VEL
LIN {X 0,Y 320.219,Z 393.281,A -85,B 0,C 180,E1 -15804.295,E2 -15804.295} C_VEL
LIN {X 0,Y 322.755,Z 382.281,A -85,B 0,C 180,E1 -15806.391,E2 -15806.391} C_VEL
LIN {X 0,Y 325.364,Z 370.249,A -85,B 0,C 180,E1 -15808.266,E2 -15808.266} C_VEL
LIN {X 0,Y 327.884,Z 357.148,A -85,B 0,C 180,E1 -15809.935,E2 -15809.935} C_VEL
LIN {X 0,Y 330.076,Z 344.536,A -85,B 0,C 180,E1 -15811.237,E2 -15811.237} C_VEL
LIN {X 0,Y 331.401,Z 335.539,A -85,B 0,C 180,E1 -15812.019,E2 -15812.019} C_VEL
LIN {X 0,Y 331.075,Z 332.573,A -85,B 0,C 180,E1 -15812.333,E2 -15812.333} C_VEL
LIN {X 0,Y 327.556,Z 320.22,A -85,B 0,C 180,E1 -15813.792,E2 -15813.792} C_VEL
LIN {X 0,Y 322.717,Z 307.168,A -85,B 0,C 180,E1 -15815.286,E2 -15815.286} C_VEL
LIN {X 0,Y 322.015,Z 305.587,A -85,B 0,C 180,E1 -15815.468,E2 -15815.468} C_VEL
LIN {X 0,Y 320.173,Z 302.909,A -85,B 0,C 180,E1 -15815.87,E2 -15815.87} C_VEL
LIN {X 0,Y 316.01,Z 299.781,A -85,B 0,C 180,E1 -15816.625,E2 -15816.625} C_VEL
LIN {X 0,Y 310.835,Z 296.093,A -85,B 0,C 180,E1 -15817.552,E2 -15817.552} C_VEL
LIN {X 0,Y 309.435,Z 294.38,A -85,B 0,C 180,E1 -15817.834,E2 -15817.834} C_VEL
LIN {X 0,Y 307.591,Z 291.035,A -85,B 0,C 180,E1 -15818.251,E2 -15818.251} C_VEL
LIN {X 0,Y 306.127,Z 288.482,A -85,B 0,C 180,E1 -15818.584,E2 -15818.584} C_VEL
LIN {X 0,Y 305.77,Z 287.041,A -85,B 0,C 180,E1 -15818.734,E2 -15818.734} C_VEL
LIN {X 0,Y 305.868,Z 285.703,A -85,B 0,C 180,E1 -15821.237,E2 -15821.237} C_VEL
LIN {X 0,Y 305.874,Z 283.672,A -85,B 0,C 180,E1 -15825.362,E2 -15825.362} C_VEL
LIN {X 0,Y 305.632,Z 282.04,A -85,B 0,C 180,E1 -15829.401,E2 -15829.401} C_VEL
LIN {X 0,Y 305.807,Z 282.018,A -85,B 0,C 180,E1 -15832.076,E2 -15832.076} C_VEL
LIN {X 0,Y 305.685,Z 282.033,A -85,B 0,C 180,E1 -15834.725,E2 -15834.725} C_VEL
LIN {X 0,Y 305.953,Z 282.001,A -85,B 0,C 180,E1 -15838.685,E2 -15838.685} C_VEL
LIN {X 0,Y 305.953,Z 281.999,A -85,B 0,C 180,E1 -15841.318,E2 -15841.318} C_VEL
LIN {X 0,Y 305.849,Z 282.01,A -85,B 0,C 180,E1 -15846.599,E2 -15846.599} C_VEL
LIN {X 0,Y 305.732,Z 282.026,A -85,B 0,C 180,E1 -15849.261,E2 -15849.261} C_VEL
LIN {X 0,Y 305.585,Z 282.041,A -85,B 0,C 180,E1 -15853.297,E2 -15853.297} C_VEL
LIN {X 0,Y 305.591,Z 282.044,A -85,B 0,C 180,E1 -15856.021,E2 -15856.021} C_VEL
LIN {X 0,Y 305.574,Z 282.042,A -85,B 0,C 180,E1 -15859.447,E2 -15859.447} C_VEL
LIN {X 0,Y 305.488,Z 282.055,A -85,B 0,C 180,E1 -15863.043,E2 -15863.043} C_VEL
LIN {X 0,Y 305.506,Z 282.057,A -85,B 0,C 180,E1 -15864.463,E2 -15864.463} C_VEL
LIN {X 0,Y 305.783,Z 283.614,A -85,B 0,C 180,E1 -15867.367,E2 -15867.367} C_VEL
LIN {X 0,Y 306.096,Z 285.582,A -85,B 0,C 180,E1 -15870.341,E2 -15870.341} C_VEL
LIN {X 0,Y 306.637,Z 288.718,A -85,B 0,C 180,E1 -15874.403,E2 -15874.403} C_VEL
LIN {X 0,Y 307.222,Z 292.103,A -85,B 0,C 180,E1 -15878.146,E2 -15878.146} C_VEL
LIN {X 0,Y 307.778,Z 295.513,A -85,B 0,C 180,E1 -15881.469,E2 -15881.469} C_VEL
LIN {X 0,Y 308.499,Z 299.589,A -85,B 0,C 180,E1 -15885.073,E2 -15885.073} C_VEL
LIN {X 0,Y 308.776,Z 301.873,A -85,B 0,C 180,E1 -15886.937,E2 -15886.937} C_VEL
LIN {X 0,Y 308.395,Z 305.365,A -85,B 0,C 180,E1 -15889.527,E2 -15889.527} C_VEL
LIN {X 0,Y 307.413,Z 311.145,A -85,B 0,C 180,E1 -15893.531,E2 -15893.531} C_VEL
LIN {X 0,Y 307.207,Z 312.532,A -85,B 0,C 180,E1 -15894.463,E2 -15894.463} C_VEL
LIN {X 0,Y 308.208,Z 316.01,A -85,B 0,C 180,E1 -15894.744,E2 -15894.744} C_VEL
LIN {X 0,Y 309.062,Z 318.017,A -85,B 0,C 180,E1 -15894.949,E2 -15894.949} C_VEL
LIN {X 0,Y 314.079,Z 332.398,A -85,B 0,C 180,E1 -15896.303,E2 -15896.303} C_VEL
LIN {X 0,Y 317.2,Z 344.609,A -85,B 0,C 180,E1 -15897.457,E2 -15897.457} C_VEL
LIN {X 0,Y 319.566,Z 357.402,A -85,B 0,C 180,E1 -15898.712,E2 -15898.712} C_VEL
LIN {X 0,Y 320.87,Z 369.49,A -85,B 0,C 180,E1 -15899.951,E2 -15899.951} C_VEL
LIN {X 0,Y 321.514,Z 379.698,A -85,B 0,C 180,E1 -15901.112,E2 -15901.112} C_VEL
LIN {X 0,Y 319.171,Z 392.385,A -85,B 0,C 180,E1 -15902.458,E2 -15902.458} C_VEL
LIN {X 0,Y 316.528,Z 404.462,A -85,B 0,C 180,E1 -15903.992,E2 -15903.992} C_VEL
LIN {X 0,Y 313.803,Z 416.633,A -85,B 0,C 180,E1 -15905.876,E2 -15905.876} C_VEL
LIN {X 0,Y 311.464,Z 427.082,A -85,B 0,C 180,E1 -15907.83,E2 -15907.83} C_VEL
LIN {X 0,Y 309.273,Z 437.021,A -85,B 0,C 180,E1 -15910.072,E2 -15910.072} C_VEL
LIN {X 0,Y 307.384,Z 445.457,A -85,B 0,C 180,E1 -15912.366,E2 -15912.366} C_VEL
LIN {X 0,Y 305.769,Z 453.052,A -85,B 0,C 180,E1 -15914.877,E2 -15914.877} C_VEL
LIN {X 0,Y 304.834,Z 459.097,A -85,B 0,C 180,E1 -15917.349,E2 -15917.349} C_VEL
LIN {X 0,Y 304.126,Z 464.275,A -85,B 0,C 180,E1 -15920.02,E2 -15920.02} C_VEL
LIN {X 0,Y 303.871,Z 467.312,A -85,B 0,C 180,E1 -15922.024,E2 -15922.024} C_VEL
LIN {X 0,Y 303.767,Z 470.228,A -85,B 0,C 180,E1 -15924.691,E2 -15924.691} C_VEL
LIN {X 0,Y 303.712,Z 471.945,A -85,B 0,C 180,E1 -15927.348,E2 -15927.348} C_VEL
LIN {X 0,Y 303.82,Z 472.499,A -85,B 0,C 180,E1 -15930.001,E2 -15930.001} C_VEL
LIN {X 0,Y 303.709,Z 471.859,A -85,B 0,C 180,E1 -15932.654,E2 -15932.654} C_VEL
LIN {X 0,Y 303.759,Z 469.983,A -85,B 0,C 180,E1 -15935.311,E2 -15935.311} C_VEL
LIN {X 0,Y 303.893,Z 466.882,A -85,B 0,C 180,E1 -15937.977,E2 -15937.977} C_VEL
LIN {X 0,Y 304.243,Z 462.495,A -85,B 0,C 180,E1 -15940.65,E2 -15940.65} C_VEL
LIN {X 0,Y 305.034,Z 456.717,A -85,B 0,C 180,E1 -15943.322,E2 -15943.322} C_VEL
LIN {X 0,Y 306.277,Z 449.398,A -85,B 0,C 180,E1 -15945.984,E2 -15945.984} C_VEL
LIN {X 0,Y 307.779,Z 441.57,A -85,B 0,C 180,E1 -15948.3,E2 -15948.3} C_VEL
LIN {X 0,Y 309.819,Z 432.175,A -85,B 0,C 180,E1 -15950.586,E2 -15950.586} C_VEL
LIN {X 0,Y 311.693,Z 422.615,A -85,B 0,C 180,E1 -15952.54,E2 -15952.54} C_VEL
LIN {X 0,Y 314.096,Z 411.298,A -85,B 0,C 180,E1 -15954.454,E2 -15954.454} C_VEL
LIN {X 0,Y 316.459,Z 398.884,A -85,B 0,C 180,E1 -15956.193,E2 -15956.193} C_VEL
LIN {X 0,Y 318.825,Z 386.722,A -85,B 0,C 180,E1 -15957.576,E2 -15957.576} C_VEL
LIN {X 0,Y 320.148,Z 378.067,A -85,B 0,C 180,E1 -15958.43,E2 -15958.43} C_VEL
LIN {X 0,Y 318.457,Z 363.851,A -85,B 0,C 180,E1 -15959.91,E2 -15959.91} C_VEL
LIN {X 0,Y 316.034,Z 349.816,A -85,B 0,C 180,E1 -15961.19,E2 -15961.19} C_VEL
LIN {X 0,Y 312.363,Z 333.984,A -85,B 0,C 180,E1 -15962.464,E2 -15962.464} C_VEL
LIN {X 0,Y 307.714,Z 318.528,A -85,B 0,C 180,E1 -15963.565,E2 -15963.565} C_VEL
LIN {X 0,Y 306.817,Z 315.191,A -85,B 0,C 180,E1 -15963.795,E2 -15963.795} C_VEL
LIN {X 0,Y 307.527,Z 310.387,A -85,B 0,C 180,E1 -15966.882,E2 -15966.882} C_VEL
LIN {X 0,Y 308.355,Z 304.948,A -85,B 0,C 180,E1 -15970.465,E2 -15970.465} C_VEL
LIN {X 0,Y 308.64,Z 300.981,A -85,B 0,C 180,E1 -15973.224,E2 -15973.224} C_VEL
LIN {X 0,Y 308.177,Z 297.382,A -85,B 0,C 180,E1 -15975.927,E2 -15975.927} C_VEL
LIN {X 0,Y 307.446,Z 293.549,A -85,B 0,C 180,E1 -15978.97,E2 -15978.97} C_VEL
LIN {X 0,Y 306.573,Z 288.277,A -85,B 0,C 180,E1 -15983.412,E2 -15983.412} C_VEL
LIN {X 0,Y 305.979,Z 284.852,A -85,B 0,C 180,E1 -15986.546,E2 -15986.546} C_VEL
LIN {X 0,Y 305.477,Z 282.06,A -85,B 0,C 180,E1 -15989.264,E2 -15989.264} C_VEL
LIN {X 0,Y 305.521,Z 282.056,A -85,B 0,C 180,E1 -15992.607,E2 -15992.607} C_VEL
LIN {X 0,Y 305.514,Z 282.054,A -85,B 0,C 180,E1 -15995.538,E2 -15995.538} C_VEL
LIN {X 0,Y 305.526,Z 282.051,A -85,B 0,C 180,E1 -15999.814,E2 -15999.814} C_VEL
LIN {X 0,Y 305.581,Z 282.048,A -85,B 0,C 180,E1 -16002.602,E2 -16002.602} C_VEL
LIN {X 0,Y 305.655,Z 282.035,A -85,B 0,C 180,E1 -16005.348,E2 -16005.348} C_VEL
LIN {X 0,Y 305.641,Z 282.037,A -85,B 0,C 180,E1 -16009.399,E2 -16009.399} C_VEL
LIN {X 0,Y 305.769,Z 282.023,A -85,B 0,C 180,E1 -16012.072,E2 -16012.072} C_VEL
LIN {X 0,Y 305.679,Z 282.034,A -85,B 0,C 180,E1 -16014.722,E2 -16014.722} C_VEL
LIN {X 0,Y 305.962,Z 281.999,A -85,B 0,C 180,E1 -16018.682,E2 -16018.682} C_VEL
LIN {X 0,Y 305.961,Z 281.995,A -85,B 0,C 180,E1 -16021.315,E2 -16021.315} C_VEL
LIN {X 0,Y 305.853,Z 282.011,A -85,B 0,C 180,E1 -16026.628,E2 -16026.628} C_VEL
LIN {X 0,Y 305.739,Z 282.022,A -85,B 0,C 180,E1 -16029.258,E2 -16029.258} C_VEL
LIN {X 0,Y 305.591,Z 282.037,A -85,B 0,C 180,E1 -16033.294,E2 -16033.294} C_VEL
LIN {X 0,Y 305.596,Z 282.044,A -85,B 0,C 180,E1 -16036.018,E2 -16036.018} C_VEL
LIN {X 0,Y 305.578,Z 282.039,A -85,B 0,C 180,E1 -16039.443,E2 -16039.443} C_VEL
LIN {X 0,Y 305.491,Z 282.054,A -85,B 0,C 180,E1 -16043.039,E2 -16043.039} C_VEL
LIN {X 0,Y 305.531,Z 282.049,A -85,B 0,C 180,E1 -16046.219,E2 -16046.219} C_VEL
LIN {X 0,Y 305.487,Z 282.05,A -85,B 0,C 180,E1 -16049.045,E2 -16049.045} C_VEL
LIN {X 0,Y 305.442,Z 282.065,A -85,B 0,C 180,E1 -16051.95,E2 -16051.95} C_VEL
LIN {X 0,Y 305.46,Z 282.054,A -85,B 0,C 180,E1 -16055.111,E2 -16055.111} C_VEL
LIN {X 0,Y 305.464,Z 282.058,A -85,B 0,C 180,E1 -16058.531,E2 -16058.531} C_VEL
LIN {X 0,Y 305.482,Z 282.05,A -85,B 0,C 180,E1 -16062.59,E2 -16062.59} C_VEL
LIN {X 0,Y 305.492,Z 282.055,A -85,B 0,C 180,E1 -16066.356,E2 -16066.356} C_VEL
LIN {X 0,Y 305.495,Z 282.054,A -85,B 0,C 180,E1 -16069.897,E2 -16069.897} C_VEL
LIN {X 0,Y 305.496,Z 282.057,A -85,B 0,C 180,E1 -16073.624,E2 -16073.624} C_VEL
LIN {X 0,Y 305.458,Z 282.059,A -85,B 0,C 180,E1 -16076.481,E2 -16076.481} C_VEL
LIN {X 0,Y 305.496,Z 282.053,A -85,B 0,C 180,E1 -16080.946,E2 -16080.946} C_VEL
LIN {X 0,Y 305.565,Z 282.045,A -85,B 0,C 180,E1 -16084.086,E2 -16084.086} C_VEL
LIN {X 0,Y 305.492,Z 282.054,A -85,B 0,C 180,E1 -16088.401,E2 -16088.401} C_VEL
LIN {X 0,Y 305.582,Z 282.047,A -85,B 0,C 180,E1 -16091.216,E2 -16091.216} C_VEL
LIN {X 0,Y 305.64,Z 282.039,A -85,B 0,C 180,E1 -16095.348,E2 -16095.348} C_VEL
LIN {X 0,Y 305.631,Z 282.041,A -85,B 0,C 180,E1 -16099.399,E2 -16099.399} C_VEL
LIN {X 0,Y 305.802,Z 282.009,A -85,B 0,C 180,E1 -16102.073,E2 -16102.073} C_VEL
LIN {X 0,Y 305.837,Z 282.01,A -85,B 0,C 180,E1 -16103.401,E2 -16103.401} C_VEL
LIN {X 0,Y 305.328,Z 282.08,A -85,B 0,C 180,E1 -16107.361,E2 -16107.361} C_VEL
LIN {X 0,Y 305.743,Z 282.779,A -85,B 0,C 180,E1 -16108.682,E2 -16108.682} C_VEL
LIN {X 0,Y 305.573,Z 283.352,A -85,B 0,C 180,E1 -16109.464,E2 -16109.464} C_VEL
LIN {X 0,Y 306.576,Z 286.398,A -85,B 0,C 180,E1 -16109.694,E2 -16109.694} C_VEL
LIN {X 0,Y 311.412,Z 298.517,A -85,B 0,C 180,E1 -16110.714,E2 -16110.714} C_VEL
LIN {X 0,Y 315.931,Z 310.016,A -85,B 0,C 180,E1 -16111.841,E2 -16111.841} C_VEL
LIN {X 0,Y 320.148,Z 323.77,A -85,B 0,C 180,E1 -16113.247,E2 -16113.247} C_VEL
LIN {X 0,Y 322.311,Z 333.214,A -85,B 0,C 180,E1 -16114.269,E2 -16114.269} C_VEL
LIN {X 0,Y 320.403,Z 346.86,A -85,B 0,C 180,E1 -16115.506,E2 -16115.506} C_VEL
LIN {X 0,Y 318.288,Z 359.648,A -85,B 0,C 180,E1 -16116.93,E2 -16116.93} C_VEL
LIN {X 0,Y 316.051,Z 372.155,A -85,B 0,C 180,E1 -16118.632,E2 -16118.632} C_VEL
LIN {X 0,Y 314.025,Z 382.467,A -85,B 0,C 180,E1 -16120.313,E2 -16120.313} C_VEL
LIN {X 0,Y 311.823,Z 393.004,A -85,B 0,C 180,E1 -16122.363,E2 -16122.363} C_VEL
LIN {X 0,Y 309.852,Z 401.946,A -85,B 0,C 180,E1 -16124.447,E2 -16124.447} C_VEL
LIN {X 0,Y 308.178,Z 409.997,A -85,B 0,C 180,E1 -16126.71,E2 -16126.71} C_VEL
LIN {X 0,Y 306.667,Z 417.429,A -85,B 0,C 180,E1 -16129.274,E2 -16129.274} C_VEL
LIN {X 0,Y 305.601,Z 422.819,A -85,B 0,C 180,E1 -16131.589,E2 -16131.589} C_VEL
LIN {X 0,Y 304.878,Z 426.923,A -85,B 0,C 180,E1 -16133.79,E2 -16133.79} C_VEL
LIN {X 0,Y 304.327,Z 430.212,A -85,B 0,C 180,E1 -16136.025,E2 -16136.025} C_VEL
LIN {X 0,Y 303.801,Z 433.255,A -85,B 0,C 180,E1 -16139.064,E2 -16139.064} C_VEL
LIN {X 0,Y 303.669,Z 434.398,A -85,B 0,C 180,E1 -16141.099,E2 -16141.099} C_VEL
LIN {X 0,Y 303.652,Z 434.947,A -85,B 0,C 180,E1 -16143.742,E2 -16143.742} C_VEL
LIN {X 0,Y 303.735,Z 434.542,A -85,B 0,C 180,E1 -16145.922,E2 -16145.922} C_VEL
LIN {X 0,Y 304.098,Z 432.993,A -85,B 0,C 180,E1 -16148.607,E2 -16148.607} C_VEL
LIN {X 0,Y 304.504,Z 431.317,A -85,B 0,C 180,E1 -16150.394,E2 -16150.394} C_VEL
LIN {X 0,Y 305.12,Z 428.604,A -85,B 0,C 180,E1 -16152.52,E2 -16152.52} C_VEL
LIN {X 0,Y 305.879,Z 425.184,A -85,B 0,C 180,E1 -16154.583,E2 -16154.583} C_VEL
LIN {X 0,Y 307.161,Z 419.953,A -85,B 0,C 180,E1 -16157.068,E2 -16157.068} C_VEL
LIN {X 0,Y 308.865,Z 413.046,A -85,B 0,C 180,E1 -16159.663,E2 -16159.663} C_VEL
LIN {X 0,Y 311.071,Z 404.399,A -85,B 0,C 180,E1 -16162.254,E2 -16162.254} C_VEL
LIN {X 0,Y 313.392,Z 394.965,A -85,B 0,C 180,E1 -16164.549,E2 -16164.549} C_VEL
LIN {X 0,Y 315.562,Z 386.024,A -85,B 0,C 180,E1 -16166.357,E2 -16166.357} C_VEL
LIN {X 0,Y 318.218,Z 374.635,A -85,B 0,C 180,E1 -16168.271,E2 -16168.271} C_VEL
LIN {X 0,Y 320.801,Z 362.155,A -85,B 0,C 180,E1 -16170.001,E2 -16170.001} C_VEL
LIN {X 0,Y 323.149,Z 349.706,A -85,B 0,C 180,E1 -16171.417,E2 -16171.417} C_VEL
LIN {X 0,Y 325.263,Z 336.585,A -85,B 0,C 180,E1 -16172.635,E2 -16172.635} C_VEL
LIN {X 0,Y 322.136,Z 324.488,A -85,B 0,C 180,E1 -16174.131,E2 -16174.131} C_VEL
LIN {X 0,Y 317.354,Z 310.937,A -85,B 0,C 180,E1 -16175.773,E2 -16175.773} C_VEL
LIN {X 0,Y 311.701,Z 298.723,A -85,B 0,C 180,E1 -16177.278,E2 -16177.278} C_VEL
LIN {X 0,Y 309.435,Z 294.38,A -85,B 0,C 180,E1 -16177.834,E2 -16177.834} C_VEL
LIN {X 0,Y 307.193,Z 291.849,A -85,B 0,C 180,E1 -16178.281,E2 -16178.281} C_VEL
LIN {X 0,Y 303.769,Z 289.532,A -85,B 0,C 180,E1 -16178.981,E2 -16178.981} C_VEL
LIN {X 0,Y 300.725,Z 288.075,A -85,B 0,C 180,E1 -16179.805,E2 -16179.805} C_VEL
LIN {X 0,Y 299.222,Z 287.375,A -85,B 0,C 180,E1 -16180.515,E2 -16180.515} C_VEL
LIN {X 0,Y 298.868,Z 287.057,A -85,B 0,C 180,E1 -16181.023,E2 -16181.023} C_VEL
LIN {X 0,Y 298.916,Z 285.127,A -85,B 0,C 180,E1 -16185.013,E2 -16185.013} C_VEL
LIN {X 0,Y 298.664,Z 283.421,A -85,B 0,C 180,E1 -16189.151,E2 -16189.151} C_VEL
LIN {X 0,Y 298.754,Z 282.896,A -85,B 0,C 180,E1 -16191.116,E2 -16191.116} C_VEL
LIN {X 0,Y 298.792,Z 282.893,A -85,B 0,C 180,E1 -16193.248,E2 -16193.248} C_VEL
LIN {X 0,Y 298.919,Z 282.876,A -85,B 0,C 180,E1 -16198.654,E2 -16198.654} C_VEL
